LIN {X 0,Y 420.408,Z 179.012,A -85,B 0,C 180,E1 -10010.808,E2 -10010.808} C_VEL
LIN {X 0,Y 420.567,Z 173.267,A -85,B 0,C 180,E1 -10012.086,E2 -10012.086} C_VEL
LIN {X 0,Y 418.323,Z 161.696,A -85,B 0,C 180,E1 -10014.875,E2 -10014.875} C_VEL
LIN {X 0,Y 418.291,Z 161.388,A -85,B 0,C 180,E1 -10015.076,E2 -10015.076} C_VEL
LIN {X 0,Y 418.293,Z 161.379,A -85,B 0,C 180,E1 -10018.063,E2 -10018.063} C_VEL
LIN {X 0,Y 418.212,Z 161.381,A -85,B 0,C 180,E1 -10021.396,E2 -10021.396} C_VEL
LIN {X 0,Y 418.266,Z 161.374,A -85,B 0,C 180,E1 -10024.58,E2 -10024.58} C_VEL
LIN {X 0,Y 418.226,Z 161.39,A -85,B 0,C 180,E1 -10027.833,E2 -10027.833} C_VEL
LIN {X 0,Y 418.221,Z 161.38,A -85,B 0,C 180,E1 -10030.948,E2 -10030.948} C_VEL
LIN {X 0,Y 418.208,Z 161.391,A -85,B 0,C 180,E1 -10033.729,E2 -10033.729} C_VEL
LIN {X 0,Y 418.206,Z 161.372,A -85,B 0,C 180,E1 -10036.448,E2 -10036.448} C_VEL
LIN {X 0,Y 418.222,Z 161.384,A -85,B 0,C 180,E1 -10039.129,E2 -10039.129} C_VEL
LIN {X 0,Y 418.227,Z 161.383,A -85,B 0,C 180,E1 -10042.166,E2 -10042.166} C_VEL
LIN {X 0,Y 418.262,Z 161.354,A -85,B 0,C 180,E1 -10045.419,E2 -10045.419} C_VEL
LIN {X 0,Y 418.208,Z 161.389,A -85,B 0,C 180,E1 -10048.603,E2 -10048.603} C_VEL
LIN {X 0,Y 418.287,Z 161.376,A -85,B 0,C 180,E1 -10051.936,E2 -10051.936} C_VEL
LIN {X 0,Y 418.285,Z 161.379,A -85,B 0,C 180,E1 -10055.162,E2 -10055.162} C_VEL
LIN {X 0,Y 418.228,Z 161.382,A -85,B 0,C 180,E1 -10058.303,E2 -10058.303} C_VEL
LIN {X 0,Y 418.278,Z 161.382,A -85,B 0,C 180,E1 -10061.383,E2 -10061.383} C_VEL
LIN {X 0,Y 418.296,Z 161.369,A -85,B 0,C 180,E1 -10064.406,E2 -10064.406} C_VEL
LIN {X 0,Y 418.349,Z 161.372,A -85,B 0,C 180,E1 -10067.385,E2 -10067.385} C_VEL
LIN {X 0,Y 418.334,Z 161.361,A -85,B 0,C 180,E1 -10070.328,E2 -10070.328} C_VEL
LIN {X 0,Y 418.507,Z 161.348,A -85,B 0,C 180,E1 -10072.279,E2 -10072.279} C_VEL
LIN {X 0,Y 418.502,Z 161.352,A -85,B 0,C 180,E1 -10074.217,E2 -10074.217} C_VEL
LIN {X 0,Y 418.534,Z 161.342,A -85,B 0,C 180,E1 -10078.075,E2 -10078.075} C_VEL
LIN {X 0,Y 418.663,Z 161.333,A -85,B 0,C 180,E1 -10080,E2 -10080} C_VEL
LIN {X 0,Y 418.492,Z 161.352,A -85,B 0,C 180,E1 -10082.888,E2 -10082.888} C_VEL
LIN {X 0,Y 418.497,Z 161.352,A -85,B 0,C 180,E1 -10085.783,E2 -10085.783} C_VEL
LIN {X 0,Y 418.371,Z 161.368,A -85,B 0,C 180,E1 -10088.696,E2 -10088.696} C_VEL
LIN {X 0,Y 418.308,Z 161.37,A -85,B 0,C 180,E1 -10091.631,E2 -10091.631} C_VEL
LIN {X 0,Y 418.296,Z 161.377,A -85,B 0,C 180,E1 -10094.597,E2 -10094.597} C_VEL
LIN {X 0,Y 418.273,Z 161.374,A -85,B 0,C 180,E1 -10097.604,E2 -10097.604} C_VEL
LIN {X 0,Y 418.244,Z 161.384,A -85,B 0,C 180,E1 -10100.663,E2 -10100.663} C_VEL
LIN {X 0,Y 418.269,Z 161.374,A -85,B 0,C 180,E1 -10103.782,E2 -10103.782} C_VEL
LIN {X 0,Y 418.306,Z 161.382,A -85,B 0,C 180,E1 -10107.071,E2 -10107.071} C_VEL
LIN {X 0,Y 418.24,Z 161.38,A -85,B 0,C 180,E1 -10110.273,E2 -10110.273} C_VEL
LIN {X 0,Y 418.243,Z 161.38,A -85,B 0,C 180,E1 -10113.678,E2 -10113.678} C_VEL
LIN {X 0,Y 418.236,Z 161.366,A -85,B 0,C 180,E1 -10117.225,E2 -10117.225} C_VEL
LIN {X 0,Y 418.24,Z 161.384,A -85,B 0,C 180,E1 -10119.683,E2 -10119.683} C_VEL
LIN {X 0,Y 418.22,Z 161.386,A -85,B 0,C 180,E1 -10122.321,E2 -10122.321} C_VEL
LIN {X 0,Y 418.233,Z 161.39,A -85,B 0,C 180,E1 -10125.109,E2 -10125.109} C_VEL
LIN {X 0,Y 418.221,Z 161.386,A -85,B 0,C 180,E1 -10127.765,E2 -10127.765} C_VEL
LIN {X 0,Y 418.236,Z 161.372,A -85,B 0,C 180,E1 -10131.557,E2 -10131.557} C_VEL
LIN {X 0,Y 418.258,Z 161.379,A -85,B 0,C 180,E1 -10135.159,E2 -10135.159} C_VEL
LIN {X 0,Y 418.245,Z 161.387,A -85,B 0,C 180,E1 -10137.472,E2 -10137.472} C_VEL
LIN {X 0,Y 418.263,Z 161.386,A -85,B 0,C 180,E1 -10140.897,E2 -10140.897} C_VEL
LIN {X 0,Y 418.285,Z 161.441,A -85,B 0,C 180,E1 -10143.695,E2 -10143.695} C_VEL
LIN {X 0,Y 420.231,Z 171.346,A -85,B 0,C 180,E1 -10146.074,E2 -10146.074} C_VEL
LIN {X 0,Y 420.944,Z 175.757,A -85,B 0,C 180,E1 -10147.079,E2 -10147.079} C_VEL
LIN {X 0,Y 420.015,Z 190.491,A -85,B 0,C 180,E1 -10150.21,E2 -10150.21} C_VEL
LIN {X 0,Y 419.851,Z 194.089,A -85,B 0,C 180,E1 -10150.917,E2 -10150.917} C_VEL
LIN {X 0,Y 422.242,Z 207.63,A -85,B 0,C 180,E1 -10151.3,E2 -10151.3} C_VEL
LIN {X 0,Y 423.878,Z 217.834,A -85,B 0,C 180,E1 -10151.553,E2 -10151.553} C_VEL
LIN {X 0,Y 422.982,Z 301.78,A -85,B 0,C 180,E1 -10153.003,E2 -10153.003} C_VEL
LIN {X 0,Y 422.43,Z 315.009,A -85,B 0,C 180,E1 -10153.415,E2 -10153.415} C_VEL
LIN {X 0,Y 421.891,Z 327.144,A -85,B 0,C 180,E1 -10153.984,E2 -10153.984} C_VEL
LIN {X 0,Y 421.162,Z 339.385,A -85,B 0,C 180,E1 -10154.762,E2 -10154.762} C_VEL
LIN {X 0,Y 420.427,Z 350.645,A -85,B 0,C 180,E1 -10155.696,E2 -10155.696} C_VEL
LIN {X 0,Y 419.714,Z 361.373,A -85,B 0,C 180,E1 -10156.812,E2 -10156.812} C_VEL
LIN {X 0,Y 419.06,Z 369.887,A -85,B 0,C 180,E1 -10157.899,E2 -10157.899} C_VEL
LIN {X 0,Y 418.446,Z 377.741,A -85,B 0,C 180,E1 -10159.108,E2 -10159.108} C_VEL
LIN {X 0,Y 417.882,Z 385.409,A -85,B 0,C 180,E1 -10160.562,E2 -10160.562} C_VEL
LIN {X 0,Y 417.432,Z 392.477,A -85,B 0,C 180,E1 -10162.259,E2 -10162.259} C_VEL
LIN {X 0,Y 417.239,Z 396.897,A -85,B 0,C 180,E1 -10163.618,E2 -10163.618} C_VEL
LIN {X 0,Y 417.146,Z 400.769,A -85,B 0,C 180,E1 -10165.167,E2 -10165.167} C_VEL
LIN {X 0,Y 417.016,Z 402.62,A -85,B 0,C 180,E1 -10166.134,E2 -10166.134} C_VEL
LIN {X 0,Y 417.031,Z 404.999,A -85,B 0,C 180,E1 -10168.068,E2 -10168.068} C_VEL
LIN {X 0,Y 416.982,Z 405.818,A -85,B 0,C 180,E1 -10170,E2 -10170} C_VEL
LIN {X 0,Y 417.031,Z 404.997,A -85,B 0,C 180,E1 -10171.931,E2 -10171.931} C_VEL
LIN {X 0,Y 417.016,Z 402.616,A -85,B 0,C 180,E1 -10173.865,E2 -10173.865} C_VEL
LIN {X 0,Y 417.167,Z 399.693,A -85,B 0,C 180,E1 -10175.316,E2 -10175.316} C_VEL
LIN {X 0,Y 417.316,Z 395.735,A -85,B 0,C 180,E1 -10176.77,E2 -10176.77} C_VEL
LIN {X 0,Y 417.616,Z 389.647,A -85,B 0,C 180,E1 -10178.467,E2 -10178.467} C_VEL
LIN {X 0,Y 418.044,Z 382.993,A -85,B 0,C 180,E1 -10179.922,E2 -10179.922} C_VEL
LIN {X 0,Y 418.643,Z 374.734,A -85,B 0,C 180,E1 -10181.376,E2 -10181.376} C_VEL
LIN {X 0,Y 419.337,Z 366.267,A -85,B 0,C 180,E1 -10182.584,E2 -10182.584} C_VEL
LIN {X 0,Y 420.064,Z 355.745,A -85,B 0,C 180,E1 -10183.798,E2 -10183.798} C_VEL
LIN {X 0,Y 420.83,Z 344.015,A -85,B 0,C 180,E1 -10184.878,E2 -10184.878} C_VEL
LIN {X 0,Y 421.563,Z 332.157,A -85,B 0,C 180,E1 -10185.718,E2 -10185.718} C_VEL
LIN {X 0,Y 422.237,Z 319.815,A -85,B 0,C 180,E1 -10186.374,E2 -10186.374} C_VEL
LIN {X 0,Y 422.762,Z 307.137,A -85,B 0,C 180,E1 -10186.85,E2 -10186.85} C_VEL
LIN {X 0,Y 423.082,Z 293.853,A -85,B 0,C 180,E1 -10187.148,E2 -10187.148} C_VEL
LIN {X 0,Y 423.755,Z 216.699,A -85,B 0,C 180,E1 -10188.465,E2 -10188.465} C_VEL
LIN {X 0,Y 419.861,Z 194.269,A -85,B 0,C 180,E1 -10189.059,E2 -10189.059} C_VEL
LIN {X 0,Y 419.935,Z 191.573,A -85,B 0,C 180,E1 -10189.554,E2 -10189.554} C_VEL
LIN {X 0,Y 420.92,Z 177.278,A -85,B 0,C 180,E1 -10192.582,E2 -10192.582} C_VEL
LIN {X 0,Y 420.491,Z 172.503,A -85,B 0,C 180,E1 -10193.648,E2 -10193.648} C_VEL
LIN {X 0,Y 418.304,Z 161.56,A -85,B 0,C 180,E1 -10196.236,E2 -10196.236} C_VEL
LIN {X 0,Y 418.257,Z 161.387,A -85,B 0,C 180,E1 -10199.161,E2 -10199.161} C_VEL
LIN {X 0,Y 418.254,Z 161.384,A -85,B 0,C 180,E1 -10202.843,E2 -10202.843} C_VEL
LIN {X 0,Y 418.239,Z 161.386,A -85,B 0,C 180,E1 -10206.237,E2 -10206.237} C_VEL
LIN {X 0,Y 418.223,Z 161.386,A -85,B 0,C 180,E1 -10209.683,E2 -10209.683} C_VEL
LIN {X 0,Y 418.217,Z 161.386,A -85,B 0,C 180,E1 -10212.319,E2 -10212.319} C_VEL
LIN {X 0,Y 418.23,Z 161.39,A -85,B 0,C 180,E1 -10215.108,E2 -10215.108} C_VEL
LIN {X 0,Y 418.233,Z 161.384,A -85,B 0,C 180,E1 -10217.766,E2 -10217.766} C_VEL
LIN {X 0,Y 418.238,Z 161.386,A -85,B 0,C 180,E1 -10220.62,E2 -10220.62} C_VEL
LIN {X 0,Y 418.234,Z 161.365,A -85,B 0,C 180,E1 -10223.975,E2 -10223.975} C_VEL
LIN {X 0,Y 418.248,Z 161.388,A -85,B 0,C 180,E1 -10227.155,E2 -10227.155} C_VEL
LIN {X 0,Y 418.259,Z 161.38,A -85,B 0,C 180,E1 -10230.895,E2 -10230.895} C_VEL
LIN {X 0,Y 418.258,Z 161.382,A -85,B 0,C 180,E1 -10234.095,E2 -10234.095} C_VEL
LIN {X 0,Y 418.22,Z 161.387,A -85,B 0,C 180,E1 -10237.263,E2 -10237.263} C_VEL
LIN {X 0,Y 418.271,Z 161.382,A -85,B 0,C 180,E1 -10240.364,E2 -10240.364} C_VEL
LIN {X 0,Y 418.304,Z 161.374,A -85,B 0,C 180,E1 -10243.404,E2 -10243.404} C_VEL
LIN {X 0,Y 418.344,Z 161.368,A -85,B 0,C 180,E1 -10246.994,E2 -10246.994} C_VEL
LIN {X 0,Y 418.332,Z 161.37,A -85,B 0,C 180,E1 -10250.328,E2 -10250.328} C_VEL
LIN {X 0,Y 418.477,Z 161.352,A -85,B 0,C 180,E1 -10253.249,E2 -10253.249} C_VEL
LIN {X 0,Y 418.324,Z 161.364,A -85,B 0,C 180,E1 -10255.181,E2 -10255.181} C_VEL
LIN {X 0,Y 418.53,Z 161.348,A -85,B 0,C 180,E1 -10258.075,E2 -10258.075} C_VEL
LIN {X 0,Y 418.659,Z 161.333,A -85,B 0,C 180,E1 -10260,E2 -10260} C_VEL
LIN {X 0,Y 418.487,Z 161.349,A -85,B 0,C 180,E1 -10262.888,E2 -10262.888} C_VEL
LIN {X 0,Y 418.478,Z 161.354,A -85,B 0,C 180,E1 -10266.751,E2 -10266.751} C_VEL
LIN {X 0,Y 418.388,Z 161.357,A -85,B 0,C 180,E1 -10268.695,E2 -10268.695} C_VEL
LIN {X 0,Y 418.304,Z 161.374,A -85,B 0,C 180,E1 -10271.631,E2 -10271.631} C_VEL
LIN {X 0,Y 418.291,Z 161.373,A -85,B 0,C 180,E1 -10274.598,E2 -10274.598} C_VEL
LIN {X 0,Y 418.277,Z 161.377,A -85,B 0,C 180,E1 -10277.604,E2 -10277.604} C_VEL
LIN {X 0,Y 418.239,Z 161.381,A -85,B 0,C 180,E1 -10280.664,E2 -10280.664} C_VEL
LIN {X 0,Y 418.278,Z 161.378,A -85,B 0,C 180,E1 -10283.782,E2 -10283.782} C_VEL
LIN {X 0,Y 418.301,Z 161.371,A -85,B 0,C 180,E1 -10287.071,E2 -10287.071} C_VEL
LIN {X 0,Y 418.235,Z 161.39,A -85,B 0,C 180,E1 -10290.273,E2 -10290.273} C_VEL
LIN {X 0,Y 418.24,Z 161.372,A -85,B 0,C 180,E1 -10293.678,E2 -10293.678} C_VEL
LIN {X 0,Y 418.232,Z 161.376,A -85,B 0,C 180,E1 -10297.225,E2 -10297.225} C_VEL
LIN {X 0,Y 418.241,Z 161.387,A -85,B 0,C 180,E1 -10299.683,E2 -10299.683} C_VEL
LIN {X 0,Y 418.222,Z 161.374,A -85,B 0,C 180,E1 -10302.322,E2 -10302.322} C_VEL
LIN {X 0,Y 418.229,Z 161.379,A -85,B 0,C 180,E1 -10305.11,E2 -10305.11} C_VEL
LIN {X 0,Y 418.234,Z 161.388,A -85,B 0,C 180,E1 -10307.768,E2 -10307.768} C_VEL
LIN {X 0,Y 418.24,Z 161.374,A -85,B 0,C 180,E1 -10310.622,E2 -10310.622} C_VEL
LIN {X 0,Y 418.24,Z 161.383,A -85,B 0,C 180,E1 -10313.977,E2 -10313.977} C_VEL
LIN {X 0,Y 418.255,Z 161.385,A -85,B 0,C 180,E1 -10317.157,E2 -10317.157} C_VEL
LIN {X 0,Y 418.267,Z 161.383,A -85,B 0,C 180,E1 -10320.897,E2 -10320.897} C_VEL
LIN {X 0,Y 418.269,Z 161.383,A -85,B 0,C 180,E1 -10324.097,E2 -10324.097} C_VEL
LIN {X 0,Y 418.289,Z 161.528,A -85,B 0,C 180,E1 -10325.164,E2 -10325.164} C_VEL
LIN {X 0,Y 420.482,Z 172.831,A -85,B 0,C 180,E1 -10327.911,E2 -10327.911} C_VEL
LIN {X 0,Y 420.548,Z 176.275,A -85,B 0,C 180,E1 -10328.687,E2 -10328.687} C_VEL
LIN {X 0,Y 419.948,Z 186.936,A -85,B 0,C 180,E1 -10330.972,E2 -10330.972} C_VEL
LIN {X 0,Y 421.24,Z 194.005,A -85,B 0,C 180,E1 -10331.195,E2 -10331.195} C_VEL
LIN {X 0,Y 423.914,Z 208.785,A -85,B 0,C 180,E1 -10331.578,E2 -10331.578} C_VEL
LIN {X 0,Y 423.001,Z 294.776,A -85,B 0,C 180,E1 -10333.067,E2 -10333.067} C_VEL
LIN {X 0,Y 422.592,Z 307.097,A -85,B 0,C 180,E1 -10333.454,E2 -10333.454} C_VEL
LIN {X 0,Y 421.954,Z 319.914,A -85,B 0,C 180,E1 -10334.049,E2 -10334.049} C_VEL
LIN {X 0,Y 421.314,Z 331.29,A -85,B 0,C 180,E1 -10334.769,E2 -10334.769} C_VEL
LIN {X 0,Y 420.637,Z 342.748,A -85,B 0,C 180,E1 -10335.712,E2 -10335.712} C_VEL
LIN {X 0,Y 419.925,Z 353.455,A -85,B 0,C 180,E1 -10336.819,E2 -10336.819} C_VEL
LIN {X 0,Y 419.231,Z 362.024,A -85,B 0,C 180,E1 -10337.905,E2 -10337.905} C_VEL
LIN {X 0,Y 418.653,Z 369.918,A -85,B 0,C 180,E1 -10339.115,E2 -10339.115} C_VEL
LIN {X 0,Y 418.129,Z 376.948,A -85,B 0,C 180,E1 -10340.425,E2 -10340.425} C_VEL
LIN {X 0,Y 417.298,Z 380.14,A -85,B 0,C 180,E1 -10341.099,E2 -10341.099} C_VEL
LIN {X 0,Y 414.13,Z 384.851,A -85,B 0,C 180,E1 -10342.219,E2 -10342.219} C_VEL
LIN {X 0,Y 410.989,Z 388.898,A -85,B 0,C 180,E1 -10343.402,E2 -10343.402} C_VEL
LIN {X 0,Y 410.217,Z 390.994,A -85,B 0,C 180,E1 -10344.167,E2 -10344.167} C_VEL
LIN {X 0,Y 410.126,Z 393.124,A -85,B 0,C 180,E1 -10345.085,E2 -10345.085} C_VEL
LIN {X 0,Y 409.982,Z 394.993,A -85,B 0,C 180,E1 -10346.069,E2 -10346.069} C_VEL
LIN {X 0,Y 409.952,Z 396.401,A -85,B 0,C 180,E1 -10347.052,E2 -10347.052} C_VEL
LIN {X 0,Y 409.971,Z 397.401,A -85,B 0,C 180,E1 -10348.036,E2 -10348.036} C_VEL
LIN {X 0,Y 409.907,Z 398.253,A -85,B 0,C 180,E1 -10350,E2 -10350} C_VEL
LIN {X 0,Y 409.92,Z 398.064,A -85,B 0,C 180,E1 -10350.983,E2 -10350.983} C_VEL
LIN {X 0,Y 409.971,Z 397.477,A -85,B 0,C 180,E1 -10351.965,E2 -10351.965} C_VEL
LIN {X 0,Y 409.979,Z 395.145,A -85,B 0,C 180,E1 -10353.932,E2 -10353.932} C_VEL
LIN {X 0,Y 410.166,Z 392.267,A -85,B 0,C 180,E1 -10355.408,E2 -10355.408} C_VEL
LIN {X 0,Y 410.347,Z 388.366,A -85,B 0,C 180,E1 -10356.886,E2 -10356.886} C_VEL
LIN {X 0,Y 410.618,Z 383.335,A -85,B 0,C 180,E1 -10358.365,E2 -10358.365} C_VEL
LIN {X 0,Y 411.124,Z 377.002,A -85,B 0,C 180,E1 -10359.843,E2 -10359.843} C_VEL
LIN {X 0,Y 411.71,Z 369.077,A -85,B 0,C 180,E1 -10361.321,E2 -10361.321} C_VEL
LIN {X 0,Y 412.541,Z 359.221,A -85,B 0,C 180,E1 -10362.795,E2 -10362.795} C_VEL
LIN {X 0,Y 413.278,Z 349.771,A -85,B 0,C 180,E1 -10363.929,E2 -10363.929} C_VEL
LIN {X 0,Y 413.976,Z 338.643,A -85,B 0,C 180,E1 -10365.005,E2 -10365.005} C_VEL
LIN {X 0,Y 414.802,Z 327.443,A -85,B 0,C 180,E1 -10365.855,E2 -10365.855} C_VEL
LIN {X 0,Y 415.4,Z 316.084,A -85,B 0,C 180,E1 -10366.526,E2 -10366.526} C_VEL
LIN {X 0,Y 415.978,Z 303.133,A -85,B 0,C 180,E1 -10367.071,E2 -10367.071} C_VEL
LIN {X 0,Y 416.339,Z 289.288,A -85,B 0,C 180,E1 -10367.435,E2 -10367.435} C_VEL
LIN {X 0,Y 417.045,Z 208.536,A -85,B 0,C 180,E1 -10368.841,E2 -10368.841} C_VEL
LIN {X 0,Y 413.049,Z 187.174,A -85,B 0,C 180,E1 -10369.443,E2 -10369.443} C_VEL
LIN {X 0,Y 413.47,Z 180.22,A -85,B 0,C 180,E1 -10370.913,E2 -10370.913} C_VEL
LIN {X 0,Y 413.742,Z 175.616,A -85,B 0,C 180,E1 -10371.944,E2 -10371.944} C_VEL
LIN {X 0,Y 411.652,Z 164.315,A -85,B 0,C 180,E1 -10374.687,E2 -10374.687} C_VEL
LIN {X 0,Y 411.241,Z 162.288,A -85,B 0,C 180,E1 -10375.273,E2 -10375.273} C_VEL
LIN {X 0,Y 411.26,Z 162.258,A -85,B 0,C 180,E1 -10377.477,E2 -10377.477} C_VEL
LIN {X 0,Y 411.19,Z 162.257,A -85,B 0,C 180,E1 -10380.847,E2 -10380.847} C_VEL
LIN {X 0,Y 411.206,Z 162.255,A -85,B 0,C 180,E1 -10384.333,E2 -10384.333} C_VEL
LIN {X 0,Y 411.191,Z 162.266,A -85,B 0,C 180,E1 -10387.973,E2 -10387.973} C_VEL
LIN {X 0,Y 411.162,Z 162.258,A -85,B 0,C 180,E1 -10391.228,E2 -10391.228} C_VEL
LIN {X 0,Y 411.174,Z 162.262,A -85,B 0,C 180,E1 -10394.49,E2 -10394.49} C_VEL
LIN {X 0,Y 411.175,Z 162.256,A -85,B 0,C 180,E1 -10398.194,E2 -10398.194} C_VEL
LIN {X 0,Y 411.219,Z 162.259,A -85,B 0,C 180,E1 -10400.776,E2 -10400.776} C_VEL
LIN {X 0,Y 411.195,Z 162.233,A -85,B 0,C 180,E1 -10404.471,E2 -10404.471} C_VEL
LIN {X 0,Y 411.204,Z 162.251,A -85,B 0,C 180,E1 -10406.873,E2 -10406.873} C_VEL
LIN {X 0,Y 411.229,Z 162.256,A -85,B 0,C 180,E1 -10410.644,E2 -10410.644} C_VEL
LIN {X 0,Y 411.232,Z 162.255,A -85,B 0,C 180,E1 -10413.619,E2 -10413.619} C_VEL
LIN {X 0,Y 411.19,Z 162.259,A -85,B 0,C 180,E1 -10416.852,E2 -10416.852} C_VEL
LIN {X 0,Y 411.21,Z 162.264,A -85,B 0,C 180,E1 -10420.05,E2 -10420.05} C_VEL
LIN {X 0,Y 411.258,Z 162.252,A -85,B 0,C 180,E1 -10423.131,E2 -10423.131} C_VEL
LIN {X 0,Y 411.3,Z 162.247,A -85,B 0,C 180,E1 -10426.896,E2 -10426.896} C_VEL
LIN {X 0,Y 411.286,Z 162.24,A -85,B 0,C 180,E1 -10430.161,E2 -10430.161} C_VEL
LIN {X 0,Y 411.476,Z 162.225,A -85,B 0,C 180,E1 -10432.146,E2 -10432.146} C_VEL
LIN {X 0,Y 411.464,Z 162.229,A -85,B 0,C 180,E1 -10434.118,E2 -10434.118} C_VEL
LIN {X 0,Y 411.503,Z 162.217,A -85,B 0,C 180,E1 -10438.042,E2 -10438.042} C_VEL
LIN {X 0,Y 411.632,Z 162.209,A -85,B 0,C 180,E1 -10440,E2 -10440} C_VEL
LIN {X 0,Y 411.449,Z 162.23,A -85,B 0,C 180,E1 -10442.937,E2 -10442.937} C_VEL
LIN {X 0,Y 411.458,Z 162.228,A -85,B 0,C 180,E1 -10445.882,E2 -10445.882} C_VEL
LIN {X 0,Y 411.312,Z 162.248,A -85,B 0,C 180,E1 -10448.846,E2 -10448.846} C_VEL
LIN {X 0,Y 411.277,Z 162.247,A -85,B 0,C 180,E1 -10451.833,E2 -10451.833} C_VEL
LIN {X 0,Y 411.253,Z 162.256,A -85,B 0,C 180,E1 -10454.853,E2 -10454.853} C_VEL
LIN {X 0,Y 411.239,Z 162.249,A -85,B 0,C 180,E1 -10457.916,E2 -10457.916} C_VEL
LIN {X 0,Y 411.19,Z 162.266,A -85,B 0,C 180,E1 -10461.034,E2 -10461.034} C_VEL
LIN {X 0,Y 411.206,Z 162.253,A -85,B 0,C 180,E1 -10464.217,E2 -10464.217} C_VEL
LIN {X 0,Y 411.254,Z 162.256,A -85,B 0,C 180,E1 -10467.478,E2 -10467.478} C_VEL
LIN {X 0,Y 411.185,Z 162.263,A -85,B 0,C 180,E1 -10470.848,E2 -10470.848} C_VEL
LIN {X 0,Y 411.2,Z 162.256,A -85,B 0,C 180,E1 -10474.334,E2 -10474.334} C_VEL
LIN {X 0,Y 411.188,Z 162.251,A -85,B 0,C 180,E1 -10477.975,E2 -10477.975} C_VEL
LIN {X 0,Y 411.157,Z 162.269,A -85,B 0,C 180,E1 -10481.228,E2 -10481.228} C_VEL
LIN {X 0,Y 411.173,Z 162.265,A -85,B 0,C 180,E1 -10484.491,E2 -10484.491} C_VEL
LIN {X 0,Y 411.162,Z 162.266,A -85,B 0,C 180,E1 -10488.193,E2 -10488.193} C_VEL
LIN {X 0,Y 411.181,Z 162.255,A -85,B 0,C 180,E1 -10490.772,E2 -10490.772} C_VEL
LIN {X 0,Y 411.196,Z 162.267,A -85,B 0,C 180,E1 -10494.472,E2 -10494.472} C_VEL
LIN {X 0,Y 411.207,Z 162.258,A -85,B 0,C 180,E1 -10496.874,E2 -10496.874} C_VEL
LIN {X 0,Y 411.212,Z 162.265,A -85,B 0,C 180,E1 -10500.65,E2 -10500.65} C_VEL
LIN {X 0,Y 411.273,Z 162.44,A -85,B 0,C 180,E1 -10503.489,E2 -10503.489} C_VEL
LIN {X 0,Y 413.754,Z 175.101,A -85,B 0,C 180,E1 -10506.527,E2 -10506.527} C_VEL
LIN {X 0,Y 413.998,Z 178.443,A -85,B 0,C 180,E1 -10507.282,E2 -10507.282} C_VEL
LIN {X 0,Y 412.963,Z 194.027,A -85,B 0,C 180,E1 -10510.587,E2 -10510.587} C_VEL
LIN {X 0,Y 416.04,Z 211.615,A -85,B 0,C 180,E1 -10511.083,E2 -10511.083} C_VEL
LIN {X 0,Y 417.134,Z 219.006,A -85,B 0,C 180,E1 -10511.266,E2 -10511.266} C_VEL
LIN {X 0,Y 416.213,Z 301.727,A -85,B 0,C 180,E1 -10512.718,E2 -10512.718} C_VEL
LIN {X 0,Y 415.636,Z 314.952,A -85,B 0,C 180,E1 -10513.136,E2 -10513.136} C_VEL
LIN {X 0,Y 415.081,Z 327.085,A -85,B 0,C 180,E1 -10513.714,E2 -10513.714} C_VEL
LIN {X 0,Y 414.307,Z 339.324,A -85,B 0,C 180,E1 -10514.504,E2 -10514.504} C_VEL
LIN {X 0,Y 413.541,Z 350.579,A -85,B 0,C 180,E1 -10515.452,E2 -10515.452} C_VEL
LIN {X 0,Y 412.778,Z 361.311,A -85,B 0,C 180,E1 -10516.586,E2 -10516.586} C_VEL
LIN {X 0,Y 412.102,Z 369.825,A -85,B 0,C 180,E1 -10517.691,E2 -10517.691} C_VEL
LIN {X 0,Y 411.428,Z 377.677,A -85,B 0,C 180,E1 -10518.92,E2 -10518.92} C_VEL
LIN {X 0,Y 410.859,Z 385.345,A -85,B 0,C 180,E1 -10520.399,E2 -10520.399} C_VEL
LIN {X 0,Y 410.378,Z 392.413,A -85,B 0,C 180,E1 -10522.125,E2 -10522.125} C_VEL
LIN {X 0,Y 410.133,Z 397.276,A -85,B 0,C 180,E1 -10523.661,E2 -10523.661} C_VEL
LIN {X 0,Y 410.058,Z 400.705,A -85,B 0,C 180,E1 -10525.084,E2 -10525.084} C_VEL
LIN {X 0,Y 409.936,Z 402.556,A -85,B 0,C 180,E1 -10526.067,E2 -10526.067} C_VEL
LIN {X 0,Y 409.927,Z 404.935,A -85,B 0,C 180,E1 -10528.035,E2 -10528.035} C_VEL
LIN {X 0,Y 409.918,Z 405.539,A -85,B 0,C 180,E1 -10529.017,E2 -10529.017} C_VEL
LIN {X 0,Y 409.906,Z 405.753,A -85,B 0,C 180,E1 -10530,E2 -10530} C_VEL
LIN {X 0,Y 409.918,Z 405.537,A -85,B 0,C 180,E1 -10530.982,E2 -10530.982} C_VEL
LIN {X 0,Y 409.927,Z 404.932,A -85,B 0,C 180,E1 -10531.965,E2 -10531.965} C_VEL
LIN {X 0,Y 409.936,Z 402.55,A -85,B 0,C 180,E1 -10533.932,E2 -10533.932} C_VEL
LIN {X 0,Y 410.086,Z 399.627,A -85,B 0,C 180,E1 -10535.408,E2 -10535.408} C_VEL
LIN {X 0,Y 410.251,Z 395.669,A -85,B 0,C 180,E1 -10536.887,E2 -10536.887} C_VEL
LIN {X 0,Y 410.562,Z 389.58,A -85,B 0,C 180,E1 -10538.614,E2 -10538.614} C_VEL
LIN {X 0,Y 411.017,Z 382.926,A -85,B 0,C 180,E1 -10540.093,E2 -10540.093} C_VEL
LIN {X 0,Y 411.644,Z 374.667,A -85,B 0,C 180,E1 -10541.572,E2 -10541.572} C_VEL
LIN {X 0,Y 412.404,Z 366.2,A -85,B 0,C 180,E1 -10542.799,E2 -10542.799} C_VEL
LIN {X 0,Y 413.104,Z 356.439,A -85,B 0,C 180,E1 -10543.954,E2 -10543.954} C_VEL
LIN {X 0,Y 413.852,Z 345.373,A -85,B 0,C 180,E1 -10545.008,E2 -10545.008} C_VEL
LIN {X 0,Y 414.602,Z 334.012,A -85,B 0,C 180,E1 -10545.862,E2 -10545.862} C_VEL
LIN {X 0,Y 415.304,Z 322.345,A -85,B 0,C 180,E1 -10546.529,E2 -10546.529} C_VEL
LIN {X 0,Y 415.899,Z 308.893,A -85,B 0,C 180,E1 -10547.073,E2 -10547.073} C_VEL
LIN {X 0,Y 416.284,Z 295.555,A -85,B 0,C 180,E1 -10547.405,E2 -10547.405} C_VEL
LIN {X 0,Y 417.099,Z 218,A -85,B 0,C 180,E1 -10548.745,E2 -10548.745} C_VEL
LIN {X 0,Y 412.956,Z 194.35,A -85,B 0,C 180,E1 -10549.381,E2 -10549.381} C_VEL
LIN {X 0,Y 412.957,Z 192.697,A -85,B 0,C 180,E1 -10549.639,E2 -10549.639} C_VEL
LIN {X 0,Y 413.98,Z 178.402,A -85,B 0,C 180,E1 -10552.718,E2 -10552.718} C_VEL
LIN {X 0,Y 413.603,Z 174.093,A -85,B 0,C 180,E1 -10553.696,E2 -10553.696} C_VEL
LIN {X 0,Y 411.27,Z 162.413,A -85,B 0,C 180,E1 -10556.511,E2 -10556.511} C_VEL
LIN {X 0,Y 411.195,Z 162.263,A -85,B 0,C 180,E1 -10559.712,E2 -10559.712} C_VEL
LIN {X 0,Y 411.203,Z 162.258,A -85,B 0,C 180,E1 -10563.155,E2 -10563.155} C_VEL
LIN {X 0,Y 411.187,Z 162.266,A -85,B 0,C 180,E1 -10566.551,E2 -10566.551} C_VEL
LIN {X 0,Y 411.19,Z 162.262,A -85,B 0,C 180,E1 -10569.724,E2 -10569.724} C_VEL
LIN {X 0,Y 411.165,Z 162.266,A -85,B 0,C 180,E1 -10573.133,E2 -10573.133} C_VEL
LIN {X 0,Y 411.161,Z 162.264,A -85,B 0,C 180,E1 -10575.88,E2 -10575.88} C_VEL
LIN {X 0,Y 411.156,Z 162.269,A -85,B 0,C 180,E1 -10578.771,E2 -10578.771} C_VEL
LIN {X 0,Y 411.184,Z 162.25,A -85,B 0,C 180,E1 -10582.025,E2 -10582.025} C_VEL
LIN {X 0,Y 411.196,Z 162.257,A -85,B 0,C 180,E1 -10585.665,E2 -10585.665} C_VEL
LIN {X 0,Y 411.179,Z 162.263,A -85,B 0,C 180,E1 -10589.151,E2 -10589.151} C_VEL
LIN {X 0,Y 411.249,Z 162.256,A -85,B 0,C 180,E1 -10592.522,E2 -10592.522} C_VEL
LIN {X 0,Y 411.2,Z 162.252,A -85,B 0,C 180,E1 -10595.783,E2 -10595.783} C_VEL
LIN {X 0,Y 411.185,Z 162.267,A -85,B 0,C 180,E1 -10598.965,E2 -10598.965} C_VEL
LIN {X 0,Y 411.234,Z 162.249,A -85,B 0,C 180,E1 -10602.084,E2 -10602.084} C_VEL
LIN {X 0,Y 411.25,Z 162.257,A -85,B 0,C 180,E1 -10605.147,E2 -10605.147} C_VEL
LIN {X 0,Y 411.288,Z 162.245,A -85,B 0,C 180,E1 -10608.167,E2 -10608.167} C_VEL
LIN {X 0,Y 411.429,Z 162.235,A -85,B 0,C 180,E1 -10612.189,E2 -10612.189} C_VEL
LIN {X 0,Y 411.458,Z 162.228,A -85,B 0,C 180,E1 -10614.118,E2 -10614.118} C_VEL
LIN {X 0,Y 411.499,Z 162.224,A -85,B 0,C 180,E1 -10618.043,E2 -10618.043} C_VEL
LIN {X 0,Y 411.628,Z 162.209,A -85,B 0,C 180,E1 -10620,E2 -10620} C_VEL
LIN {X 0,Y 411.444,Z 162.226,A -85,B 0,C 180,E1 -10622.937,E2 -10622.937} C_VEL
LIN {X 0,Y 411.446,Z 162.229,A -85,B 0,C 180,E1 -10626.867,E2 -10626.867} C_VEL
LIN {X 0,Y 411.342,Z 162.233,A -85,B 0,C 180,E1 -10628.846,E2 -10628.846} C_VEL
LIN {X 0,Y 411.272,Z 162.251,A -85,B 0,C 180,E1 -10631.833,E2 -10631.833} C_VEL
LIN {X 0,Y 411.248,Z 162.248,A -85,B 0,C 180,E1 -10634.853,E2 -10634.853} C_VEL
LIN {X 0,Y 411.242,Z 162.255,A -85,B 0,C 180,E1 -10637.916,E2 -10637.916} C_VEL
LIN {X 0,Y 411.186,Z 162.257,A -85,B 0,C 180,E1 -10641.035,E2 -10641.035} C_VEL
LIN {X 0,Y 411.218,Z 162.263,A -85,B 0,C 180,E1 -10644.216,E2 -10644.216} C_VEL
LIN {X 0,Y 411.249,Z 162.25,A -85,B 0,C 180,E1 -10647.479,E2 -10647.479} C_VEL
LIN {X 0,Y 411.18,Z 162.264,A -85,B 0,C 180,E1 -10650.849,E2 -10650.849} C_VEL
LIN {X 0,Y 411.197,Z 162.238,A -85,B 0,C 180,E1 -10654.335,E2 -10654.335} C_VEL
LIN {X 0,Y 411.187,Z 162.26,A -85,B 0,C 180,E1 -10657.975,E2 -10657.975} C_VEL
LIN {X 0,Y 411.157,Z 162.265,A -85,B 0,C 180,E1 -10661.229,E2 -10661.229} C_VEL
LIN {X 0,Y 411.169,Z 162.256,A -85,B 0,C 180,E1 -10664.492,E2 -10664.492} C_VEL
LIN {X 0,Y 411.172,Z 162.262,A -85,B 0,C 180,E1 -10668.196,E2 -10668.196} C_VEL
LIN {X 0,Y 411.206,Z 162.251,A -85,B 0,C 180,E1 -10670.776,E2 -10670.776} C_VEL
LIN {X 0,Y 411.195,Z 162.255,A -85,B 0,C 180,E1 -10674.472,E2 -10674.472} C_VEL
LIN {X 0,Y 411.204,Z 162.262,A -85,B 0,C 180,E1 -10676.874,E2 -10676.874} C_VEL
LIN {X 0,Y 411.231,Z 162.26,A -85,B 0,C 180,E1 -10680.645,E2 -10680.645} C_VEL
LIN {X 0,Y 411.236,Z 162.258,A -85,B 0,C 180,E1 -10683.62,E2 -10683.62} C_VEL
LIN {X 0,Y 411.239,Z 162.46,A -85,B 0,C 180,E1 -10684.926,E2 -10684.926} C_VEL
LIN {X 0,Y 413.303,Z 172.889,A -85,B 0,C 180,E1 -10687.506,E2 -10687.506} C_VEL
LIN {X 0,Y 413.725,Z 176.333,A -85,B 0,C 180,E1 -10688.318,E2 -10688.318} C_VEL
LIN {X 0,Y 413.052,Z 187.056,A -85,B 0,C 180,E1 -10690.647,E2 -10690.647} C_VEL
LIN {X 0,Y 415.677,Z 200.949,A -85,B 0,C 180,E1 -10691.057,E2 -10691.057} C_VEL
LIN {X 0,Y 417.194,Z 210.215,A -85,B 0,C 180,E1 -10691.294,E2 -10691.294} C_VEL
LIN {X 0,Y 416.213,Z 294.858,A -85,B 0,C 180,E1 -10692.782,E2 -10692.782} C_VEL
LIN {X 0,Y 415.805,Z 307.173,A -85,B 0,C 180,E1 -10693.176,E2 -10693.176} C_VEL
LIN {X 0,Y 415.154,Z 319.987,A -85,B 0,C 180,E1 -10693.781,E2 -10693.781} C_VEL
LIN {X 0,Y 414.47,Z 331.361,A -85,B 0,C 180,E1 -10694.511,E2 -10694.511} C_VEL
LIN {X 0,Y 413.789,Z 341.958,A -85,B 0,C 180,E1 -10695.387,E2 -10695.387} C_VEL
LIN {X 0,Y 413.106,Z 352.456,A -85,B 0,C 180,E1 -10696.473,E2 -10696.473} C_VEL
LIN {X 0,Y 412.288,Z 362.092,A -85,B 0,C 180,E1 -10697.698,E2 -10697.698} C_VEL
LIN {X 0,Y 411.648,Z 369.986,A -85,B 0,C 180,E1 -10698.927,E2 -10698.927} C_VEL
LIN {X 0,Y 411.067,Z 377.704,A -85,B 0,C 180,E1 -10700.405,E2 -10700.405} C_VEL
LIN {X 0,Y 410.523,Z 384.789,A -85,B 0,C 180,E1 -10702.129,E2 -10702.129} C_VEL
LIN {X 0,Y 410.291,Z 389.1,A -85,B 0,C 180,E1 -10703.466,E2 -10703.466} C_VEL
LIN {X 0,Y 410.217,Z 390.994,A -85,B 0,C 180,E1 -10704.167,E2 -10704.167} C_VEL
LIN {X 0,Y 409.48,Z 392.861,A -85,B 0,C 180,E1 -10704.945,E2 -10704.945} C_VEL
LIN {X 0,Y 406.508,Z 395.32,A -85,B 0,C 180,E1 -10706.227,E2 -10706.227} C_VEL
LIN {X 0,Y 404.017,Z 396.758,A -85,B 0,C 180,E1 -10707.279,E2 -10707.279} C_VEL
LIN {X 0,Y 402.939,Z 397.545,A -85,B 0,C 180,E1 -10708.101,E2 -10708.101} C_VEL
LIN {X 0,Y 402.847,Z 397.701,A -85,B 0,C 180,E1 -10708.381,E2 -10708.381} C_VEL
LIN {X 0,Y 402.832,Z 398.318,A -85,B 0,C 180,E1 -10710,E2 -10710} C_VEL
LIN {X 0,Y 402.848,Z 398.129,A -85,B 0,C 180,E1 -10711,E2 -10711} C_VEL
LIN {X 0,Y 402.869,Z 397.542,A -85,B 0,C 180,E1 -10712,E2 -10712} C_VEL
LIN {X 0,Y 402.901,Z 395.209,A -85,B 0,C 180,E1 -10714.001,E2 -10714.001} C_VEL
LIN {X 0,Y 403.092,Z 392.331,A -85,B 0,C 180,E1 -10715.503,E2 -10715.503} C_VEL
LIN {X 0,Y 403.285,Z 388.43,A -85,B 0,C 180,E1 -10717.007,E2 -10717.007} C_VEL
LIN {X 0,Y 403.592,Z 383.398,A -85,B 0,C 180,E1 -10718.512,E2 -10718.512} C_VEL
LIN {X 0,Y 404.113,Z 377.065,A -85,B 0,C 180,E1 -10720.016,E2 -10720.016} C_VEL
LIN {X 0,Y 404.719,Z 369.14,A -85,B 0,C 180,E1 -10721.52,E2 -10721.52} C_VEL
LIN {X 0,Y 405.616,Z 359.282,A -85,B 0,C 180,E1 -10723.018,E2 -10723.018} C_VEL
LIN {X 0,Y 406.349,Z 350.147,A -85,B 0,C 180,E1 -10724.137,E2 -10724.137} C_VEL
LIN {X 0,Y 407.021,Z 340.127,A -85,B 0,C 180,E1 -10725.139,E2 -10725.139} C_VEL
LIN {X 0,Y 407.824,Z 329.265,A -85,B 0,C 180,E1 -10726.005,E2 -10726.005} C_VEL
LIN {X 0,Y 408.557,Z 317.271,A -85,B 0,C 180,E1 -10726.746,E2 -10726.746} C_VEL
LIN {X 0,Y 409.142,Z 304.984,A -85,B 0,C 180,E1 -10727.301,E2 -10727.301} C_VEL
LIN {X 0,Y 409.557,Z 292.34,A -85,B 0,C 180,E1 -10727.669,E2 -10727.669} C_VEL
LIN {X 0,Y 410.325,Z 209.43,A -85,B 0,C 180,E1 -10729.146,E2 -10729.146} C_VEL
LIN {X 0,Y 406.157,Z 187.245,A -85,B 0,C 180,E1 -10729.786,E2 -10729.786} C_VEL
LIN {X 0,Y 406.223,Z 184.89,A -85,B 0,C 180,E1 -10730.244,E2 -10730.244} C_VEL
LIN {X 0,Y 406.788,Z 176.822,A -85,B 0,C 180,E1 -10732.072,E2 -10732.072} C_VEL
LIN {X 0,Y 404.591,Z 165.109,A -85,B 0,C 180,E1 -10734.969,E2 -10734.969} C_VEL
LIN {X 0,Y 404.208,Z 163.161,A -85,B 0,C 180,E1 -10735.549,E2 -10735.549} C_VEL
LIN {X 0,Y 404.197,Z 163.135,A -85,B 0,C 180,E1 -10737.999,E2 -10737.999} C_VEL
LIN {X 0,Y 404.14,Z 163.134,A -85,B 0,C 180,E1 -10741.558,E2 -10741.558} C_VEL
LIN {X 0,Y 404.185,Z 163.126,A -85,B 0,C 180,E1 -10745.016,E2 -10745.016} C_VEL
LIN {X 0,Y 404.15,Z 163.133,A -85,B 0,C 180,E1 -10748.757,E2 -10748.757} C_VEL
LIN {X 0,Y 404.121,Z 163.136,A -85,B 0,C 180,E1 -10751.599,E2 -10751.599} C_VEL
LIN {X 0,Y 404.143,Z 163.137,A -85,B 0,C 180,E1 -10754.521,E2 -10754.521} C_VEL
LIN {X 0,Y 404.134,Z 163.123,A -85,B 0,C 180,E1 -10757.295,E2 -10757.295} C_VEL
LIN {X 0,Y 404.167,Z 163.14,A -85,B 0,C 180,E1 -10759.955,E2 -10759.955} C_VEL
LIN {X 0,Y 404.134,Z 163.132,A -85,B 0,C 180,E1 -10763.125,E2 -10763.125} C_VEL
LIN {X 0,Y 404.141,Z 163.121,A -85,B 0,C 180,E1 -10766.187,E2 -10766.187} C_VEL
LIN {X 0,Y 404.142,Z 163.144,A -85,B 0,C 180,E1 -10769.714,E2 -10769.714} C_VEL
LIN {X 0,Y 404.19,Z 163.128,A -85,B 0,C 180,E1 -10773.122,E2 -10773.122} C_VEL
LIN {X 0,Y 404.169,Z 163.139,A -85,B 0,C 180,E1 -10775.334,E2 -10775.334} C_VEL
LIN {X 0,Y 404.133,Z 163.136,A -85,B 0,C 180,E1 -10778.58,E2 -10778.58} C_VEL
LIN {X 0,Y 404.204,Z 163.137,A -85,B 0,C 180,E1 -10781.762,E2 -10781.762} C_VEL
LIN {X 0,Y 404.2,Z 163.123,A -85,B 0,C 180,E1 -10784.882,E2 -10784.882} C_VEL
LIN {X 0,Y 404.25,Z 163.128,A -85,B 0,C 180,E1 -10787.958,E2 -10787.958} C_VEL
LIN {X 0,Y 404.428,Z 163.103,A -85,B 0,C 180,E1 -10792.1,E2 -10792.1} C_VEL
LIN {X 0,Y 404.413,Z 163.108,A -85,B 0,C 180,E1 -10794.015,E2 -10794.015} C_VEL
LIN {X 0,Y 404.472,Z 163.093,A -85,B 0,C 180,E1 -10798.008,E2 -10798.008} C_VEL
LIN {X 0,Y 404.602,Z 163.085,A -85,B 0,C 180,E1 -10800,E2 -10800} C_VEL
LIN {X 0,Y 404.407,Z 163.107,A -85,B 0,C 180,E1 -10802.988,E2 -10802.988} C_VEL
LIN {X 0,Y 404.405,Z 163.106,A -85,B 0,C 180,E1 -10805.985,E2 -10805.985} C_VEL
LIN {X 0,Y 404.259,Z 163.128,A -85,B 0,C 180,E1 -10809.002,E2 -10809.002} C_VEL
LIN {X 0,Y 404.249,Z 163.121,A -85,B 0,C 180,E1 -10812.042,E2 -10812.042} C_VEL
LIN {X 0,Y 404.199,Z 163.138,A -85,B 0,C 180,E1 -10815.118,E2 -10815.118} C_VEL
LIN {X 0,Y 404.198,Z 163.125,A -85,B 0,C 180,E1 -10818.239,E2 -10818.239} C_VEL
LIN {X 0,Y 404.132,Z 163.145,A -85,B 0,C 180,E1 -10821.42,E2 -10821.42} C_VEL
LIN {X 0,Y 404.165,Z 163.131,A -85,B 0,C 180,E1 -10824.666,E2 -10824.666} C_VEL
LIN {X 0,Y 404.191,Z 163.132,A -85,B 0,C 180,E1 -10828,E2 -10828} C_VEL
LIN {X 0,Y 404.135,Z 163.144,A -85,B 0,C 180,E1 -10831.558,E2 -10831.558} C_VEL
LIN {X 0,Y 404.179,Z 163.121,A -85,B 0,C 180,E1 -10835.017,E2 -10835.017} C_VEL
LIN {X 0,Y 404.147,Z 163.132,A -85,B 0,C 180,E1 -10838.758,E2 -10838.758} C_VEL
LIN {X 0,Y 404.116,Z 163.143,A -85,B 0,C 180,E1 -10841.599,E2 -10841.599} C_VEL
LIN {X 0,Y 404.142,Z 163.141,A -85,B 0,C 180,E1 -10844.522,E2 -10844.522} C_VEL
LIN {X 0,Y 404.122,Z 163.143,A -85,B 0,C 180,E1 -10847.294,E2 -10847.294} C_VEL
LIN {X 0,Y 404.131,Z 163.14,A -85,B 0,C 180,E1 -10849.951,E2 -10849.951} C_VEL
LIN {X 0,Y 404.133,Z 163.142,A -85,B 0,C 180,E1 -10853.126,E2 -10853.126} C_VEL
LIN {X 0,Y 404.145,Z 163.133,A -85,B 0,C 180,E1 -10856.188,E2 -10856.188} C_VEL
LIN {X 0,Y 404.144,Z 163.137,A -85,B 0,C 180,E1 -10859.715,E2 -10859.715} C_VEL
LIN {X 0,Y 404.204,Z 163.277,A -85,B 0,C 180,E1 -10863.194,E2 -10863.194} C_VEL
LIN {X 0,Y 406.483,Z 174.778,A -85,B 0,C 180,E1 -10866.023,E2 -10866.023} C_VEL
LIN {X 0,Y 407.078,Z 179.57,A -85,B 0,C 180,E1 -10867.142,E2 -10867.142} C_VEL
LIN {X 0,Y 406.043,Z 193.964,A -85,B 0,C 180,E1 -10870.242,E2 -10870.242} C_VEL
LIN {X 0,Y 408.872,Z 209.861,A -85,B 0,C 180,E1 -10870.707,E2 -10870.707} C_VEL
LIN {X 0,Y 410.412,Z 219.887,A -85,B 0,C 180,E1 -10870.964,E2 -10870.964} C_VEL
LIN {X 0,Y 409.457,Z 301.675,A -85,B 0,C 180,E1 -10872.423,E2 -10872.423} C_VEL
LIN {X 0,Y 408.861,Z 314.896,A -85,B 0,C 180,E1 -10872.848,E2 -10872.848} C_VEL
LIN {X 0,Y 408.255,Z 327.026,A -85,B 0,C 180,E1 -10873.434,E2 -10873.434} C_VEL
LIN {X 0,Y 407.474,Z 339.263,A -85,B 0,C 180,E1 -10874.237,E2 -10874.237} C_VEL
LIN {X 0,Y 406.652,Z 350.54,A -85,B 0,C 180,E1 -10875.202,E2 -10875.202} C_VEL
LIN {X 0,Y 405.829,Z 361.249,A -85,B 0,C 180,E1 -10876.352,E2 -10876.352} C_VEL
LIN {X 0,Y 405.141,Z 369.762,A -85,B 0,C 180,E1 -10877.476,E2 -10877.476} C_VEL
LIN {X 0,Y 404.44,Z 377.614,A -85,B 0,C 180,E1 -10878.726,E2 -10878.726} C_VEL
LIN {X 0,Y 403.837,Z 385.281,A -85,B 0,C 180,E1 -10880.231,E2 -10880.231} C_VEL
LIN {X 0,Y 403.32,Z 392.349,A -85,B 0,C 180,E1 -10881.986,E2 -10881.986} C_VEL
LIN {X 0,Y 403.056,Z 397.54,A -85,B 0,C 180,E1 -10883.668,E2 -10883.668} C_VEL
LIN {X 0,Y 402.973,Z 400.641,A -85,B 0,C 180,E1 -10884.997,E2 -10884.997} C_VEL
LIN {X 0,Y 402.859,Z 402.491,A -85,B 0,C 180,E1 -10885.998,E2 -10885.998} C_VEL
LIN {X 0,Y 402.824,Z 404.87,A -85,B 0,C 180,E1 -10888,E2 -10888} C_VEL
LIN {X 0,Y 402.845,Z 405.475,A -85,B 0,C 180,E1 -10889,E2 -10889} C_VEL
LIN {X 0,Y 402.832,Z 405.689,A -85,B 0,C 180,E1 -10890,E2 -10890} C_VEL
LIN {X 0,Y 402.845,Z 405.472,A -85,B 0,C 180,E1 -10890.999,E2 -10890.999} C_VEL
LIN {X 0,Y 402.824,Z 404.867,A -85,B 0,C 180,E1 -10891.999,E2 -10891.999} C_VEL
LIN {X 0,Y 402.859,Z 402.485,A -85,B 0,C 180,E1 -10894.001,E2 -10894.001} C_VEL
LIN {X 0,Y 402.986,Z 399.561,A -85,B 0,C 180,E1 -10895.504,E2 -10895.504} C_VEL
LIN {X 0,Y 403.186,Z 395.603,A -85,B 0,C 180,E1 -10897.008,E2 -10897.008} C_VEL
LIN {X 0,Y 403.521,Z 389.514,A -85,B 0,C 180,E1 -10898.765,E2 -10898.765} C_VEL
LIN {X 0,Y 404.012,Z 382.859,A -85,B 0,C 180,E1 -10900.27,E2 -10900.27} C_VEL
LIN {X 0,Y 404.672,Z 374.6,A -85,B 0,C 180,E1 -10901.774,E2 -10901.774} C_VEL
LIN {X 0,Y 405.46,Z 366.132,A -85,B 0,C 180,E1 -10903.022,E2 -10903.022} C_VEL
LIN {X 0,Y 406.215,Z 355.847,A -85,B 0,C 180,E1 -10904.252,E2 -10904.252} C_VEL
LIN {X 0,Y 406.991,Z 345.304,A -85,B 0,C 180,E1 -10905.268,E2 -10905.268} C_VEL
LIN {X 0,Y 407.779,Z 333.942,A -85,B 0,C 180,E1 -10906.135,E2 -10906.135} C_VEL
LIN {X 0,Y 408.523,Z 322.273,A -85,B 0,C 180,E1 -10906.811,E2 -10906.811} C_VEL
LIN {X 0,Y 409.116,Z 308.818,A -85,B 0,C 180,E1 -10907.365,E2 -10907.365} C_VEL
LIN {X 0,Y 409.535,Z 295.472,A -85,B 0,C 180,E1 -10907.701,E2 -10907.701} C_VEL
LIN {X 0,Y 410.419,Z 219.12,A -85,B 0,C 180,E1 -10909.04,E2 -10909.04} C_VEL
LIN {X 0,Y 406.059,Z 194.277,A -85,B 0,C 180,E1 -10909.723,E2 -10909.723} C_VEL
LIN {X 0,Y 406.073,Z 192.629,A -85,B 0,C 180,E1 -10909.986,E2 -10909.986} C_VEL
LIN {X 0,Y 407.058,Z 179.527,A -85,B 0,C 180,E1 -10912.858,E2 -10912.858} C_VEL
LIN {X 0,Y 406.462,Z 174.501,A -85,B 0,C 180,E1 -10914.03,E2 -10914.03} C_VEL
LIN {X 0,Y 404.201,Z 163.262,A -85,B 0,C 180,E1 -10916.806,E2 -10916.806} C_VEL
LIN {X 0,Y 404.141,Z 163.137,A -85,B 0,C 180,E1 -10920.284,E2 -10920.284} C_VEL
LIN {X 0,Y 404.141,Z 163.134,A -85,B 0,C 180,E1 -10923.811,E2 -10923.811} C_VEL
LIN {X 0,Y 404.13,Z 163.141,A -85,B 0,C 180,E1 -10926.873,E2 -10926.873} C_VEL
LIN {X 0,Y 404.142,Z 163.139,A -85,B 0,C 180,E1 -10930.079,E2 -10930.079} C_VEL
LIN {X 0,Y 404.144,Z 163.14,A -85,B 0,C 180,E1 -10933.082,E2 -10933.082} C_VEL
LIN {X 0,Y 404.142,Z 163.138,A -85,B 0,C 180,E1 -10935.925,E2 -10935.925} C_VEL
LIN {X 0,Y 404.111,Z 163.146,A -85,B 0,C 180,E1 -10938.634,E2 -10938.634} C_VEL
LIN {X 0,Y 404.142,Z 163.129,A -85,B 0,C 180,E1 -10941.492,E2 -10941.492} C_VEL
LIN {X 0,Y 404.175,Z 163.122,A -85,B 0,C 180,E1 -10944.983,E2 -10944.983} C_VEL
LIN {X 0,Y 404.132,Z 163.145,A -85,B 0,C 180,E1 -10948.553,E2 -10948.553} C_VEL
LIN {X 0,Y 404.185,Z 163.133,A -85,B 0,C 180,E1 -10952,E2 -10952} C_VEL
LIN {X 0,Y 404.16,Z 163.131,A -85,B 0,C 180,E1 -10955.333,E2 -10955.333} C_VEL
LIN {X 0,Y 404.127,Z 163.145,A -85,B 0,C 180,E1 -10958.58,E2 -10958.58} C_VEL
LIN {X 0,Y 404.193,Z 163.125,A -85,B 0,C 180,E1 -10961.761,E2 -10961.761} C_VEL
LIN {X 0,Y 404.195,Z 163.138,A -85,B 0,C 180,E1 -10964.882,E2 -10964.882} C_VEL
LIN {X 0,Y 404.259,Z 163.119,A -85,B 0,C 180,E1 -10967.959,E2 -10967.959} C_VEL
LIN {X 0,Y 404.393,Z 163.111,A -85,B 0,C 180,E1 -10972.129,E2 -10972.129} C_VEL
LIN {X 0,Y 404.407,Z 163.105,A -85,B 0,C 180,E1 -10974.015,E2 -10974.015} C_VEL
LIN {X 0,Y 404.468,Z 163.099,A -85,B 0,C 180,E1 -10978.009,E2 -10978.009} C_VEL
LIN {X 0,Y 404.598,Z 163.085,A -85,B 0,C 180,E1 -10980,E2 -10980} C_VEL
LIN {X 0,Y 404.402,Z 163.103,A -85,B 0,C 180,E1 -10982.989,E2 -10982.989} C_VEL
LIN {X 0,Y 404.397,Z 163.106,A -85,B 0,C 180,E1 -10986.988,E2 -10986.988} C_VEL
LIN {X 0,Y 404.247,Z 163.117,A -85,B 0,C 180,E1 -10990.012,E2 -10990.012} C_VEL
LIN {X 0,Y 404.255,Z 163.125,A -85,B 0,C 180,E1 -10993.212,E2 -10993.212} C_VEL
LIN {X 0,Y 404.205,Z 163.129,A -85,B 0,C 180,E1 -10997.008,E2 -10997.008} C_VEL
LIN {X 0,Y 404.153,Z 163.139,A -85,B 0,C 180,E1 -11000.352,E2 -11000.352} C_VEL
LIN {X 0,Y 404.16,Z 163.135,A -85,B 0,C 180,E1 -11003.575,E2 -11003.575} C_VEL
LIN {X 0,Y 404.174,Z 163.139,A -85,B 0,C 180,E1 -11005.767,E2 -11005.767} C_VEL
LIN {X 0,Y 404.186,Z 163.131,A -85,B 0,C 180,E1 -11008.001,E2 -11008.001} C_VEL
LIN {X 0,Y 404.13,Z 163.143,A -85,B 0,C 180,E1 -11011.559,E2 -11011.559} C_VEL
LIN {X 0,Y 404.177,Z 163.107,A -85,B 0,C 180,E1 -11015.017,E2 -11015.017} C_VEL
LIN {X 0,Y 404.147,Z 163.14,A -85,B 0,C 180,E1 -11018.758,E2 -11018.758} C_VEL
LIN {X 0,Y 404.116,Z 163.141,A -85,B 0,C 180,E1 -11021.601,E2 -11021.601} C_VEL
LIN {X 0,Y 404.139,Z 163.132,A -85,B 0,C 180,E1 -11024.523,E2 -11024.523} C_VEL
LIN {X 0,Y 404.131,Z 163.144,A -85,B 0,C 180,E1 -11027.297,E2 -11027.297} C_VEL
LIN {X 0,Y 404.165,Z 163.124,A -85,B 0,C 180,E1 -11029.957,E2 -11029.957} C_VEL
LIN {X 0,Y 404.132,Z 163.144,A -85,B 0,C 180,E1 -11033.126,E2 -11033.126} C_VEL
LIN {X 0,Y 404.142,Z 163.14,A -85,B 0,C 180,E1 -11036.189,E2 -11036.189} C_VEL
LIN {X 0,Y 404.143,Z 163.14,A -85,B 0,C 180,E1 -11039.716,E2 -11039.716} C_VEL
LIN {X 0,Y 404.194,Z 163.137,A -85,B 0,C 180,E1 -11043.124,E2 -11043.124} C_VEL
LIN {X 0,Y 404.196,Z 163.224,A -85,B 0,C 180,E1 -11044.602,E2 -11044.602} C_VEL
LIN {X 0,Y 406.338,Z 174.145,A -85,B 0,C 180,E1 -11047.379,E2 -11047.379} C_VEL
LIN {X 0,Y 406.795,Z 177.544,A -85,B 0,C 180,E1 -11048.196,E2 -11048.196} C_VEL
LIN {X 0,Y 406.149,Z 187.124,A -85,B 0,C 180,E1 -11050.304,E2 -11050.304} C_VEL
LIN {X 0,Y 409.149,Z 202.827,A -85,B 0,C 180,E1 -11050.776,E2 -11050.776} C_VEL
LIN {X 0,Y 410.473,Z 210.573,A -85,B 0,C 180,E1 -11050.981,E2 -11050.981} C_VEL
LIN {X 0,Y 409.448,Z 294.939,A -85,B 0,C 180,E1 -11052.488,E2 -11052.488} C_VEL
LIN {X 0,Y 408.998,Z 308.01,A -85,B 0,C 180,E1 -11052.92,E2 -11052.92} C_VEL
LIN {X 0,Y 408.356,Z 320.06,A -85,B 0,C 180,E1 -11053.503,E2 -11053.503} C_VEL
LIN {X 0,Y 407.628,Z 331.432,A -85,B 0,C 180,E1 -11054.244,E2 -11054.244} C_VEL
LIN {X 0,Y 406.875,Z 342.411,A -85,B 0,C 180,E1 -11055.171,E2 -11055.171} C_VEL
LIN {X 0,Y 406.118,Z 353.592,A -85,B 0,C 180,E1 -11056.363,E2 -11056.363} C_VEL
LIN {X 0,Y 405.359,Z 362.16,A -85,B 0,C 180,E1 -11057.484,E2 -11057.484} C_VEL
LIN {X 0,Y 404.664,Z 370.053,A -85,B 0,C 180,E1 -11058.734,E2 -11058.734} C_VEL
LIN {X 0,Y 404.035,Z 377.771,A -85,B 0,C 180,E1 -11060.236,E2 -11060.236} C_VEL
LIN {X 0,Y 403.463,Z 384.855,A -85,B 0,C 180,E1 -11061.99,E2 -11061.99} C_VEL
LIN {X 0,Y 403.217,Z 389.491,A -85,B 0,C 180,E1 -11063.465,E2 -11063.465} C_VEL
LIN {X 0,Y 403.045,Z 393.19,A -85,B 0,C 180,E1 -11064.999,E2 -11064.999} C_VEL
LIN {X 0,Y 402.904,Z 395.059,A -85,B 0,C 180,E1 -11066,E2 -11066} C_VEL
LIN {X 0,Y 402.853,Z 396.466,A -85,B 0,C 180,E1 -11067,E2 -11067} C_VEL
LIN {X 0,Y 402.847,Z 397.701,A -85,B 0,C 180,E1 -11068.381,E2 -11068.381} C_VEL
LIN {X 0,Y 402.157,Z 398.189,A -85,B 0,C 180,E1 -11069.214,E2 -11069.214} C_VEL
LIN {X 0,Y 399.273,Z 398.276,A -85,B 0,C 180,E1 -11070.57,E2 -11070.57} C_VEL
LIN {X 0,Y 396.85,Z 397.873,A -85,B 0,C 180,E1 -11071.665,E2 -11071.665} C_VEL
LIN {X 0,Y 395.765,Z 397.081,A -85,B 0,C 180,E1 -11072.65,E2 -11072.65} C_VEL
LIN {X 0,Y 395.746,Z 396.886,A -85,B 0,C 180,E1 -11072.792,E2 -11072.792} C_VEL
LIN {X 0,Y 395.825,Z 395.274,A -85,B 0,C 180,E1 -11074.073,E2 -11074.073} C_VEL
LIN {X 0,Y 396.02,Z 392.395,A -85,B 0,C 180,E1 -11075.602,E2 -11075.602} C_VEL
LIN {X 0,Y 396.225,Z 388.494,A -85,B 0,C 180,E1 -11077.133,E2 -11077.133} C_VEL
LIN {X 0,Y 396.554,Z 383.461,A -85,B 0,C 180,E1 -11078.664,E2 -11078.664} C_VEL
LIN {X 0,Y 397.089,Z 377.128,A -85,B 0,C 180,E1 -11080.195,E2 -11080.195} C_VEL
LIN {X 0,Y 397.755,Z 369.202,A -85,B 0,C 180,E1 -11081.724,E2 -11081.724} C_VEL
LIN {X 0,Y 398.706,Z 359.344,A -85,B 0,C 180,E1 -11083.247,E2 -11083.247} C_VEL
LIN {X 0,Y 399.466,Z 349.895,A -85,B 0,C 180,E1 -11084.42,E2 -11084.42} C_VEL
LIN {X 0,Y 400.27,Z 338.763,A -85,B 0,C 180,E1 -11085.531,E2 -11085.531} C_VEL
LIN {X 0,Y 401.16,Z 327.56,A -85,B 0,C 180,E1 -11086.409,E2 -11086.409} C_VEL
LIN {X 0,Y 401.818,Z 316.198,A -85,B 0,C 180,E1 -11087.101,E2 -11087.101} C_VEL
LIN {X 0,Y 402.453,Z 303.237,A -85,B 0,C 180,E1 -11087.663,E2 -11087.663} C_VEL
LIN {X 0,Y 402.853,Z 289.374,A -85,B 0,C 180,E1 -11088.039,E2 -11088.039} C_VEL
LIN {X 0,Y 403.645,Z 210.372,A -85,B 0,C 180,E1 -11089.459,E2 -11089.459} C_VEL
LIN {X 0,Y 399.283,Z 187.299,A -85,B 0,C 180,E1 -11090.141,E2 -11090.141} C_VEL
LIN {X 0,Y 399.334,Z 184.95,A -85,B 0,C 180,E1 -11090.609,E2 -11090.609} C_VEL
LIN {X 0,Y 399.818,Z 178.031,A -85,B 0,C 180,E1 -11092.205,E2 -11092.205} C_VEL
LIN {X 0,Y 397.664,Z 166.543,A -85,B 0,C 180,E1 -11095.097,E2 -11095.097} C_VEL
LIN {X 0,Y 397.147,Z 164.037,A -85,B 0,C 180,E1 -11095.834,E2 -11095.834} C_VEL
LIN {X 0,Y 397.123,Z 164.014,A -85,B 0,C 180,E1 -11098.543,E2 -11098.543} C_VEL
LIN {X 0,Y 397.079,Z 164.018,A -85,B 0,C 180,E1 -11102.071,E2 -11102.071} C_VEL
LIN {X 0,Y 397.12,Z 164.007,A -85,B 0,C 180,E1 -11105.503,E2 -11105.503} C_VEL
LIN {X 0,Y 397.126,Z 164.007,A -85,B 0,C 180,E1 -11108.86,E2 -11108.86} C_VEL
LIN {X 0,Y 397.067,Z 164.022,A -85,B 0,C 180,E1 -11112.267,E2 -11112.267} C_VEL
LIN {X 0,Y 397.085,Z 164.014,A -85,B 0,C 180,E1 -11115.068,E2 -11115.068} C_VEL
LIN {X 0,Y 397.064,Z 164.01,A -85,B 0,C 180,E1 -11118.021,E2 -11118.021} C_VEL
LIN {X 0,Y 397.129,Z 164.014,A -85,B 0,C 180,E1 -11121.138,E2 -11121.138} C_VEL
LIN {X 0,Y 397.116,Z 163.985,A -85,B 0,C 180,E1 -11124.496,E2 -11124.496} C_VEL
LIN {X 0,Y 397.075,Z 164.017,A -85,B 0,C 180,E1 -11127.928,E2 -11127.928} C_VEL
LIN {X 0,Y 397.118,Z 164.016,A -85,B 0,C 180,E1 -11131.456,E2 -11131.456} C_VEL
LIN {X 0,Y 397.148,Z 164.013,A -85,B 0,C 180,E1 -11134.487,E2 -11134.487} C_VEL
LIN {X 0,Y 397.09,Z 164.013,A -85,B 0,C 180,E1 -11138.181,E2 -11138.181} C_VEL
LIN {X 0,Y 397.157,Z 164.014,A -85,B 0,C 180,E1 -11141.426,E2 -11141.426} C_VEL
LIN {X 0,Y 397.173,Z 163.998,A -85,B 0,C 180,E1 -11144.608,E2 -11144.608} C_VEL
LIN {X 0,Y 397.213,Z 164.007,A -85,B 0,C 180,E1 -11147.742,E2 -11147.742} C_VEL
LIN {X 0,Y 397.389,Z 163.98,A -85,B 0,C 180,E1 -11152.041,E2 -11152.041} C_VEL
LIN {X 0,Y 397.244,Z 163.999,A -85,B 0,C 180,E1 -11154.925,E2 -11154.925} C_VEL
LIN {X 0,Y 397.441,Z 163.968,A -85,B 0,C 180,E1 -11157.973,E2 -11157.973} C_VEL
LIN {X 0,Y 397.571,Z 163.96,A -85,B 0,C 180,E1 -11160,E2 -11160} C_VEL
LIN {X 0,Y 397.367,Z 163.985,A -85,B 0,C 180,E1 -11163.041,E2 -11163.041} C_VEL
LIN {X 0,Y 397.356,Z 163.983,A -85,B 0,C 180,E1 -11166.092,E2 -11166.092} C_VEL
LIN {X 0,Y 397.229,Z 164.005,A -85,B 0,C 180,E1 -11169.162,E2 -11169.162} C_VEL
LIN {X 0,Y 397.213,Z 163.997,A -85,B 0,C 180,E1 -11172.258,E2 -11172.258} C_VEL
LIN {X 0,Y 397.173,Z 164.012,A -85,B 0,C 180,E1 -11175.392,E2 -11175.392} C_VEL
LIN {X 0,Y 397.152,Z 164.003,A -85,B 0,C 180,E1 -11178.574,E2 -11178.574} C_VEL
LIN {X 0,Y 397.09,Z 164.018,A -85,B 0,C 180,E1 -11181.819,E2 -11181.819} C_VEL
LIN {X 0,Y 397.148,Z 164.015,A -85,B 0,C 180,E1 -11185.513,E2 -11185.513} C_VEL
LIN {X 0,Y 397.118,Z 164.014,A -85,B 0,C 180,E1 -11188.544,E2 -11188.544} C_VEL
LIN {X 0,Y 397.074,Z 164.022,A -85,B 0,C 180,E1 -11192.072,E2 -11192.072} C_VEL
LIN {X 0,Y 397.115,Z 163.994,A -85,B 0,C 180,E1 -11195.504,E2 -11195.504} C_VEL
LIN {X 0,Y 397.123,Z 164.008,A -85,B 0,C 180,E1 -11198.861,E2 -11198.861} C_VEL
LIN {X 0,Y 397.061,Z 164.021,A -85,B 0,C 180,E1 -11202.268,E2 -11202.268} C_VEL
LIN {X 0,Y 397.084,Z 164.025,A -85,B 0,C 180,E1 -11205.069,E2 -11205.069} C_VEL
LIN {X 0,Y 397.052,Z 164.023,A -85,B 0,C 180,E1 -11208.024,E2 -11208.024} C_VEL
LIN {X 0,Y 397.093,Z 164.005,A -85,B 0,C 180,E1 -11211.146,E2 -11211.146} C_VEL
LIN {X 0,Y 397.118,Z 164.021,A -85,B 0,C 180,E1 -11214.497,E2 -11214.497} C_VEL
LIN {X 0,Y 397.078,Z 164.024,A -85,B 0,C 180,E1 -11217.929,E2 -11217.929} C_VEL
LIN {X 0,Y 397.118,Z 164.017,A -85,B 0,C 180,E1 -11220.296,E2 -11220.296} C_VEL
LIN {X 0,Y 397.155,Z 164.135,A -85,B 0,C 180,E1 -11222.892,E2 -11222.892} C_VEL
LIN {X 0,Y 399.281,Z 174.73,A -85,B 0,C 180,E1 -11225.567,E2 -11225.567} C_VEL
LIN {X 0,Y 400.138,Z 180.697,A -85,B 0,C 180,E1 -11226.996,E2 -11226.996} C_VEL
LIN {X 0,Y 399.139,Z 193.902,A -85,B 0,C 180,E1 -11229.886,E2 -11229.886} C_VEL
LIN {X 0,Y 402.158,Z 210.55,A -85,B 0,C 180,E1 -11230.386,E2 -11230.386} C_VEL
LIN {X 0,Y 403.724,Z 221.54,A -85,B 0,C 180,E1 -11230.668,E2 -11230.668} C_VEL
LIN {X 0,Y 402.688,Z 301.622,A -85,B 0,C 180,E1 -11232.118,E2 -11232.118} C_VEL
LIN {X 0,Y 402.098,Z 314.84,A -85,B 0,C 180,E1 -11232.551,E2 -11232.551} C_VEL
LIN {X 0,Y 401.445,Z 326.967,A -85,B 0,C 180,E1 -11233.145,E2 -11233.145} C_VEL
LIN {X 0,Y 400.622,Z 339.202,A -85,B 0,C 180,E1 -11233.961,E2 -11233.961} C_VEL
LIN {X 0,Y 399.744,Z 350.697,A -85,B 0,C 180,E1 -11234.962,E2 -11234.962} C_VEL
LIN {X 0,Y 398.896,Z 361.186,A -85,B 0,C 180,E1 -11236.11,E2 -11236.11} C_VEL
LIN {X 0,Y 398.187,Z 369.699,A -85,B 0,C 180,E1 -11237.254,E2 -11237.254} C_VEL
LIN {X 0,Y 397.462,Z 377.551,A -85,B 0,C 180,E1 -11238.526,E2 -11238.526} C_VEL
LIN {X 0,Y 396.823,Z 385.218,A -85,B 0,C 180,E1 -11240.056,E2 -11240.056} C_VEL
LIN {X 0,Y 396.263,Z 392.285,A -85,B 0,C 180,E1 -11241.843,E2 -11241.843} C_VEL
LIN {X 0,Y 395.985,Z 397.128,A -85,B 0,C 180,E1 -11243.426,E2 -11243.426} C_VEL
LIN {X 0,Y 395.89,Z 400.576,A -85,B 0,C 180,E1 -11244.907,E2 -11244.907} C_VEL
LIN {X 0,Y 395.784,Z 402.427,A -85,B 0,C 180,E1 -11245.927,E2 -11245.927} C_VEL
LIN {X 0,Y 395.722,Z 404.805,A -85,B 0,C 180,E1 -11247.964,E2 -11247.964} C_VEL
LIN {X 0,Y 395.756,Z 405.41,A -85,B 0,C 180,E1 -11248.982,E2 -11248.982} C_VEL
LIN {X 0,Y 395.76,Z 405.624,A -85,B 0,C 180,E1 -11250,E2 -11250} C_VEL
LIN {X 0,Y 395.756,Z 405.407,A -85,B 0,C 180,E1 -11251.017,E2 -11251.017} C_VEL
LIN {X 0,Y 395.7,Z 403.809,A -85,B 0,C 180,E1 -11253.054,E2 -11253.054} C_VEL
LIN {X 0,Y 395.783,Z 402.419,A -85,B 0,C 180,E1 -11254.073,E2 -11254.073} C_VEL
LIN {X 0,Y 395.888,Z 399.495,A -85,B 0,C 180,E1 -11255.603,E2 -11255.603} C_VEL
LIN {X 0,Y 396.101,Z 395.537,A -85,B 0,C 180,E1 -11257.134,E2 -11257.134} C_VEL
LIN {X 0,Y 396.467,Z 389.447,A -85,B 0,C 180,E1 -11258.922,E2 -11258.922} C_VEL
LIN {X 0,Y 397.02,Z 382.792,A -85,B 0,C 180,E1 -11260.453,E2 -11260.453} C_VEL
LIN {X 0,Y 397.712,Z 374.533,A -85,B 0,C 180,E1 -11261.983,E2 -11261.983} C_VEL
LIN {X 0,Y 398.515,Z 366.064,A -85,B 0,C 180,E1 -11263.253,E2 -11263.253} C_VEL
LIN {X 0,Y 399.26,Z 356.567,A -85,B 0,C 180,E1 -11264.419,E2 -11264.419} C_VEL
LIN {X 0,Y 400.12,Z 345.235,A -85,B 0,C 180,E1 -11265.536,E2 -11265.536} C_VEL
LIN {X 0,Y 400.951,Z 333.872,A -85,B 0,C 180,E1 -11266.417,E2 -11266.417} C_VEL
LIN {X 0,Y 401.731,Z 322.201,A -85,B 0,C 180,E1 -11267.104,E2 -11267.104} C_VEL
LIN {X 0,Y 402.34,Z 308.743,A -85,B 0,C 180,E1 -11267.667,E2 -11267.667} C_VEL
LIN {X 0,Y 402.794,Z 295.388,A -85,B 0,C 180,E1 -11268.008,E2 -11268.008} C_VEL
LIN {X 0,Y 403.585,Z 219.266,A -85,B 0,C 180,E1 -11269.371,E2 -11269.371} C_VEL
LIN {X 0,Y 399.158,Z 194.205,A -85,B 0,C 180,E1 -11270.079,E2 -11270.079} C_VEL
LIN {X 0,Y 399.163,Z 192.561,A -85,B 0,C 180,E1 -11270.348,E2 -11270.348} C_VEL
LIN {X 0,Y 400.113,Z 180.651,A -85,B 0,C 180,E1 -11273.005,E2 -11273.005} C_VEL
LIN {X 0,Y 399.278,Z 174.682,A -85,B 0,C 180,E1 -11274.432,E2 -11274.432} C_VEL
LIN {X 0,Y 397.152,Z 164.118,A -85,B 0,C 180,E1 -11277.107,E2 -11277.107} C_VEL
LIN {X 0,Y 397.097,Z 164.017,A -85,B 0,C 180,E1 -11279.862,E2 -11279.862} C_VEL
LIN {X 0,Y 397.115,Z 164.009,A -85,B 0,C 180,E1 -11283.717,E2 -11283.717} C_VEL
LIN {X 0,Y 397.086,Z 164.013,A -85,B 0,C 180,E1 -11287.207,E2 -11287.207} C_VEL
LIN {X 0,Y 397.071,Z 164.02,A -85,B 0,C 180,E1 -11290.44,E2 -11290.44} C_VEL
LIN {X 0,Y 397.094,Z 164.02,A -85,B 0,C 180,E1 -11293.648,E2 -11293.648} C_VEL
LIN {X 0,Y 397.095,Z 164.016,A -85,B 0,C 180,E1 -11296.52,E2 -11296.52} C_VEL
LIN {X 0,Y 397.105,Z 164.017,A -85,B 0,C 180,E1 -11300.422,E2 -11300.422} C_VEL
LIN {X 0,Y 397.099,Z 163.996,A -85,B 0,C 180,E1 -11304.264,E2 -11304.264} C_VEL
LIN {X 0,Y 397.106,Z 164.016,A -85,B 0,C 180,E1 -11306.726,E2 -11306.726} C_VEL
LIN {X 0,Y 397.115,Z 164.012,A -85,B 0,C 180,E1 -11310.295,E2 -11310.295} C_VEL
LIN {X 0,Y 397.184,Z 164.009,A -85,B 0,C 180,E1 -11312.609,E2 -11312.609} C_VEL
LIN {X 0,Y 397.115,Z 164.007,A -85,B 0,C 180,E1 -11315.981,E2 -11315.981} C_VEL
LIN {X 0,Y 397.128,Z 164.013,A -85,B 0,C 180,E1 -11319.704,E2 -11319.704} C_VEL
LIN {X 0,Y 397.171,Z 164.004,A -85,B 0,C 180,E1 -11322.845,E2 -11322.845} C_VEL
LIN {X 0,Y 397.217,Z 164.003,A -85,B 0,C 180,E1 -11326.702,E2 -11326.702} C_VEL
LIN {X 0,Y 397.211,Z 163.998,A -85,B 0,C 180,E1 -11329.809,E2 -11329.809} C_VEL
LIN {X 0,Y 397.339,Z 163.988,A -85,B 0,C 180,E1 -11332.888,E2 -11332.888} C_VEL
LIN {X 0,Y 397.239,Z 163.99,A -85,B 0,C 180,E1 -11334.925,E2 -11334.925} C_VEL
LIN {X 0,Y 397.437,Z 163.975,A -85,B 0,C 180,E1 -11337.973,E2 -11337.973} C_VEL
LIN {X 0,Y 397.568,Z 163.961,A -85,B 0,C 180,E1 -11340,E2 -11340} C_VEL
LIN {X 0,Y 397.361,Z 163.979,A -85,B 0,C 180,E1 -11343.042,E2 -11343.042} C_VEL
LIN {X 0,Y 397.35,Z 163.983,A -85,B 0,C 180,E1 -11347.112,E2 -11347.112} C_VEL
LIN {X 0,Y 397.206,Z 163.996,A -85,B 0,C 180,E1 -11350.191,E2 -11350.191} C_VEL
LIN {X 0,Y 397.216,Z 164.002,A -85,B 0,C 180,E1 -11353.322,E2 -11353.322} C_VEL
LIN {X 0,Y 397.171,Z 164.005,A -85,B 0,C 180,E1 -11357.156,E2 -11357.156} C_VEL
LIN {X 0,Y 397.092,Z 164.014,A -85,B 0,C 180,E1 -11360.731,E2 -11360.731} C_VEL
LIN {X 0,Y 397.123,Z 164.015,A -85,B 0,C 180,E1 -11364.019,E2 -11364.019} C_VEL
LIN {X 0,Y 397.185,Z 164.001,A -85,B 0,C 180,E1 -11367.391,E2 -11367.391} C_VEL
LIN {X 0,Y 397.069,Z 164.022,A -85,B 0,C 180,E1 -11370.883,E2 -11370.883} C_VEL
LIN {X 0,Y 397.117,Z 163.988,A -85,B 0,C 180,E1 -11374.494,E2 -11374.494} C_VEL
LIN {X 0,Y 397.095,Z 164.019,A -85,B 0,C 180,E1 -11378.276,E2 -11378.276} C_VEL
LIN {X 0,Y 397.082,Z 164.018,A -85,B 0,C 180,E1 -11380.91,E2 -11380.91} C_VEL
LIN {X 0,Y 397.094,Z 164,A -85,B 0,C 180,E1 -11383.65,E2 -11383.65} C_VEL
LIN {X 0,Y 397.097,Z 164.02,A -85,B 0,C 180,E1 -11386.522,E2 -11386.522} C_VEL
LIN {X 0,Y 397.108,Z 164.003,A -85,B 0,C 180,E1 -11390.424,E2 -11390.424} C_VEL
LIN {X 0,Y 397.105,Z 164.011,A -85,B 0,C 180,E1 -11394.267,E2 -11394.267} C_VEL
LIN {X 0,Y 397.112,Z 164.018,A -85,B 0,C 180,E1 -11396.728,E2 -11396.728} C_VEL
LIN {X 0,Y 397.123,Z 164.019,A -85,B 0,C 180,E1 -11400.297,E2 -11400.297} C_VEL
LIN {X 0,Y 397.193,Z 164.011,A -85,B 0,C 180,E1 -11402.611,E2 -11402.611} C_VEL
LIN {X 0,Y 397.188,Z 164.226,A -85,B 0,C 180,E1 -11404.384,E2 -11404.384} C_VEL
LIN {X 0,Y 399.365,Z 175.308,A -85,B 0,C 180,E1 -11407.223,E2 -11407.223} C_VEL
LIN {X 0,Y 399.864,Z 178.757,A -85,B 0,C 180,E1 -11408.07,E2 -11408.07} C_VEL
LIN {X 0,Y 399.234,Z 187.196,A -85,B 0,C 180,E1 -11409.949,E2 -11409.949} C_VEL
LIN {X 0,Y 402.736,Z 205.19,A -85,B 0,C 180,E1 -11410.499,E2 -11410.499} C_VEL
LIN {X 0,Y 403.732,Z 211.333,A -85,B 0,C 180,E1 -11410.663,E2 -11410.663} C_VEL
LIN {X 0,Y 402.682,Z 295.02,A -85,B 0,C 180,E1 -11412.184,E2 -11412.184} C_VEL
LIN {X 0,Y 402.218,Z 308.086,A -85,B 0,C 180,E1 -11412.622,E2 -11412.622} C_VEL
LIN {X 0,Y 401.472,Z 321.237,A -85,B 0,C 180,E1 -11413.278,E2 -11413.278} C_VEL
LIN {X 0,Y 400.703,Z 333.092,A -85,B 0,C 180,E1 -11414.095,E2 -11414.095} C_VEL
LIN {X 0,Y 399.897,Z 344.3,A -85,B 0,C 180,E1 -11415.09,E2 -11415.09} C_VEL
LIN {X 0,Y 399.131,Z 354.723,A -85,B 0,C 180,E1 -11416.249,E2 -11416.249} C_VEL
LIN {X 0,Y 398.254,Z 363.927,A -85,B 0,C 180,E1 -11417.516,E2 -11417.516} C_VEL
LIN {X 0,Y 397.472,Z 372.867,A -85,B 0,C 180,E1 -11419.043,E2 -11419.043} C_VEL
LIN {X 0,Y 396.853,Z 380.065,A -85,B 0,C 180,E1 -11420.572,E2 -11420.572} C_VEL
LIN {X 0,Y 396.424,Z 384.922,A -85,B 0,C 180,E1 -11421.847,E2 -11421.847} C_VEL
LIN {X 0,Y 396.136,Z 389.907,A -85,B 0,C 180,E1 -11423.474,E2 -11423.474} C_VEL
LIN {X 0,Y 395.967,Z 393.256,A -85,B 0,C 180,E1 -11424.909,E2 -11424.909} C_VEL
LIN {X 0,Y 395.828,Z 395.124,A -85,B 0,C 180,E1 -11425.928,E2 -11425.928} C_VEL
LIN {X 0,Y 395.756,Z 396.532,A -85,B 0,C 180,E1 -11426.947,E2 -11426.947} C_VEL
LIN {X 0,Y 395.75,Z 397.781,A -85,B 0,C 180,E1 -11428.377,E2 -11428.377} C_VEL
LIN {X 0,Y 395.76,Z 398.382,A -85,B 0,C 180,E1 -11430,E2 -11430} C_VEL
LIN {X 0,Y 395.76,Z 398.193,A -85,B 0,C 180,E1 -11431.018,E2 -11431.018} C_VEL
LIN {X 0,Y 395.746,Z 396.886,A -85,B 0,C 180,E1 -11432.792,E2 -11432.792} C_VEL
LIN {X 0,Y 395.115,Z 395.948,A -85,B 0,C 180,E1 -11433.632,E2 -11433.632} C_VEL
LIN {X 0,Y 392.372,Z 393.818,A -85,B 0,C 180,E1 -11434.985,E2 -11434.985} C_VEL
LIN {X 0,Y 390.09,Z 391.605,A -85,B 0,C 180,E1 -11436.058,E2 -11436.058} C_VEL
LIN {X 0,Y 389.175,Z 389.631,A -85,B 0,C 180,E1 -11436.871,E2 -11436.871} C_VEL
LIN {X 0,Y 389.135,Z 388.886,A -85,B 0,C 180,E1 -11437.143,E2 -11437.143} C_VEL
LIN {X 0,Y 389.528,Z 383.525,A -85,B 0,C 180,E1 -11438.822,E2 -11438.822} C_VEL
LIN {X 0,Y 390.077,Z 377.191,A -85,B 0,C 180,E1 -11440.38,E2 -11440.38} C_VEL
LIN {X 0,Y 390.804,Z 369.264,A -85,B 0,C 180,E1 -11441.936,E2 -11441.936} C_VEL
LIN {X 0,Y 391.787,Z 359.406,A -85,B 0,C 180,E1 -11443.486,E2 -11443.486} C_VEL
LIN {X 0,Y 392.541,Z 349.878,A -85,B 0,C 180,E1 -11444.689,E2 -11444.689} C_VEL
LIN {X 0,Y 393.425,Z 338.823,A -85,B 0,C 180,E1 -11445.808,E2 -11445.808} C_VEL
LIN {X 0,Y 394.337,Z 327.619,A -85,B 0,C 180,E1 -11446.701,E2 -11446.701} C_VEL
LIN {X 0,Y 395.041,Z 316.254,A -85,B 0,C 180,E1 -11447.404,E2 -11447.404} C_VEL
LIN {X 0,Y 395.719,Z 303.288,A -85,B 0,C 180,E1 -11447.974,E2 -11447.974} C_VEL
LIN {X 0,Y 396.076,Z 290.922,A -85,B 0,C 180,E1 -11448.325,E2 -11448.325} C_VEL
LIN {X 0,Y 397.042,Z 211.839,A -85,B 0,C 180,E1 -11449.769,E2 -11449.769} C_VEL
LIN {X 0,Y 392.404,Z 187.354,A -85,B 0,C 180,E1 -11450.51,E2 -11450.51} C_VEL
LIN {X 0,Y 392.633,Z 183.701,A -85,B 0,C 180,E1 -11451.289,E2 -11451.289} C_VEL
LIN {X 0,Y 392.856,Z 179.24,A -85,B 0,C 180,E1 -11452.343,E2 -11452.343} C_VEL
LIN {X 0,Y 390.455,Z 166.596,A -85,B 0,C 180,E1 -11455.594,E2 -11455.594} C_VEL
LIN {X 0,Y 390.115,Z 164.908,A -85,B 0,C 180,E1 -11456.138,E2 -11456.138} C_VEL
LIN {X 0,Y 390.06,Z 164.896,A -85,B 0,C 180,E1 -11459.109,E2 -11459.109} C_VEL
LIN {X 0,Y 390.043,Z 164.901,A -85,B 0,C 180,E1 -11462.721,E2 -11462.721} C_VEL
LIN {X 0,Y 390.056,Z 164.888,A -85,B 0,C 180,E1 -11465.825,E2 -11465.825} C_VEL
LIN {X 0,Y 390.067,Z 164.884,A -85,B 0,C 180,E1 -11469.217,E2 -11469.217} C_VEL
LIN {X 0,Y 390.041,Z 164.899,A -85,B 0,C 180,E1 -11472.374,E2 -11472.374} C_VEL
LIN {X 0,Y 390.042,Z 164.891,A -85,B 0,C 180,E1 -11475.354,E2 -11475.354} C_VEL
LIN {X 0,Y 390.029,Z 164.888,A -85,B 0,C 180,E1 -11478.186,E2 -11478.186} C_VEL
LIN {X 0,Y 390.089,Z 164.891,A -85,B 0,C 180,E1 -11480.907,E2 -11480.907} C_VEL
LIN {X 0,Y 390.082,Z 164.859,A -85,B 0,C 180,E1 -11484.793,E2 -11484.793} C_VEL
LIN {X 0,Y 390.02,Z 164.901,A -85,B 0,C 180,E1 -11488.495,E2 -11488.495} C_VEL
LIN {X 0,Y 390.114,Z 164.883,A -85,B 0,C 180,E1 -11492.07,E2 -11492.07} C_VEL
LIN {X 0,Y 390.073,Z 164.896,A -85,B 0,C 180,E1 -11495.519,E2 -11495.519} C_VEL
LIN {X 0,Y 390.083,Z 164.889,A -85,B 0,C 180,E1 -11499.53,E2 -11499.53} C_VEL
LIN {X 0,Y 390.133,Z 164.884,A -85,B 0,C 180,E1 -11503.248,E2 -11503.248} C_VEL
LIN {X 0,Y 390.189,Z 164.877,A -85,B 0,C 180,E1 -11506.561,E2 -11506.561} C_VEL
LIN {X 0,Y 390.199,Z 164.864,A -85,B 0,C 180,E1 -11510.671,E2 -11510.671} C_VEL
LIN {X 0,Y 390.311,Z 164.859,A -85,B 0,C 180,E1 -11512.759,E2 -11512.759} C_VEL
LIN {X 0,Y 390.216,Z 164.874,A -85,B 0,C 180,E1 -11514.833,E2 -11514.833} C_VEL
LIN {X 0,Y 390.41,Z 164.843,A -85,B 0,C 180,E1 -11517.937,E2 -11517.937} C_VEL
LIN {X 0,Y 390.541,Z 164.836,A -85,B 0,C 180,E1 -11520,E2 -11520} C_VEL
LIN {X 0,Y 390.301,Z 164.865,A -85,B 0,C 180,E1 -11523.097,E2 -11523.097} C_VEL
LIN {X 0,Y 390.309,Z 164.861,A -85,B 0,C 180,E1 -11526.202,E2 -11526.202} C_VEL
LIN {X 0,Y 390.187,Z 164.88,A -85,B 0,C 180,E1 -11529.329,E2 -11529.329} C_VEL
LIN {X 0,Y 390.165,Z 164.875,A -85,B 0,C 180,E1 -11532.483,E2 -11532.483} C_VEL
LIN {X 0,Y 390.133,Z 164.885,A -85,B 0,C 180,E1 -11535.677,E2 -11535.677} C_VEL
LIN {X 0,Y 390.096,Z 164.884,A -85,B 0,C 180,E1 -11538.923,E2 -11538.923} C_VEL
LIN {X 0,Y 390.032,Z 164.896,A -85,B 0,C 180,E1 -11542.235,E2 -11542.235} C_VEL
LIN {X 0,Y 390.114,Z 164.889,A -85,B 0,C 180,E1 -11545.744,E2 -11545.744} C_VEL
LIN {X 0,Y 390.054,Z 164.892,A -85,B 0,C 180,E1 -11549.11,E2 -11549.11} C_VEL
LIN {X 0,Y 390.039,Z 164.901,A -85,B 0,C 180,E1 -11552.722,E2 -11552.722} C_VEL
LIN {X 0,Y 390.052,Z 164.872,A -85,B 0,C 180,E1 -11555.825,E2 -11555.825} C_VEL
LIN {X 0,Y 390.064,Z 164.892,A -85,B 0,C 180,E1 -11559.218,E2 -11559.218} C_VEL
LIN {X 0,Y 390.036,Z 164.897,A -85,B 0,C 180,E1 -11562.374,E2 -11562.374} C_VEL
LIN {X 0,Y 390.041,Z 164.899,A -85,B 0,C 180,E1 -11565.355,E2 -11565.355} C_VEL
LIN {X 0,Y 390.016,Z 164.9,A -85,B 0,C 180,E1 -11568.185,E2 -11568.185} C_VEL
LIN {X 0,Y 390.057,Z 164.883,A -85,B 0,C 180,E1 -11570.904,E2 -11570.904} C_VEL
LIN {X 0,Y 390.084,Z 164.893,A -85,B 0,C 180,E1 -11574.793,E2 -11574.793} C_VEL
LIN {X 0,Y 390.023,Z 164.901,A -85,B 0,C 180,E1 -11578.496,E2 -11578.496} C_VEL
LIN {X 0,Y 390.038,Z 164.881,A -85,B 0,C 180,E1 -11582.064,E2 -11582.064} C_VEL
LIN {X 0,Y 390.116,Z 165.165,A -85,B 0,C 180,E1 -11582.653,E2 -11582.653} C_VEL
LIN {X 0,Y 392.296,Z 175.855,A -85,B 0,C 180,E1 -11585.385,E2 -11585.385} C_VEL
LIN {X 0,Y 393.204,Z 181.824,A -85,B 0,C 180,E1 -11586.845,E2 -11586.845} C_VEL
LIN {X 0,Y 392.243,Z 193.816,A -85,B 0,C 180,E1 -11589.514,E2 -11589.514} C_VEL
LIN {X 0,Y 394.795,Z 207.518,A -85,B 0,C 180,E1 -11589.948,E2 -11589.948} C_VEL
LIN {X 0,Y 397.018,Z 221.405,A -85,B 0,C 180,E1 -11590.326,E2 -11590.326} C_VEL
LIN {X 0,Y 395.936,Z 301.57,A -85,B 0,C 180,E1 -11591.802,E2 -11591.802} C_VEL
LIN {X 0,Y 395.334,Z 314.783,A -85,B 0,C 180,E1 -11592.242,E2 -11592.242} C_VEL
LIN {X 0,Y 394.647,Z 326.908,A -85,B 0,C 180,E1 -11592.845,E2 -11592.845} C_VEL
LIN {X 0,Y 393.783,Z 339.142,A -85,B 0,C 180,E1 -11593.674,E2 -11593.674} C_VEL
LIN {X 0,Y 392.839,Z 350.969,A -85,B 0,C 180,E1 -11594.726,E2 -11594.726} C_VEL
LIN {X 0,Y 391.914,Z 362.164,A -85,B 0,C 180,E1 -11595.99,E2 -11595.99} C_VEL
LIN {X 0,Y 391.098,Z 371.308,A -85,B 0,C 180,E1 -11597.283,E2 -11597.283} C_VEL
LIN {X 0,Y 390.223,Z 380.217,A -85,B 0,C 180,E1 -11598.836,E2 -11598.836} C_VEL
LIN {X 0,Y 389.586,Z 387.384,A -85,B 0,C 180,E1 -11600.394,E2 -11600.394} C_VEL
LIN {X 0,Y 389.222,Z 392.221,A -85,B 0,C 180,E1 -11601.694,E2 -11601.694} C_VEL
LIN {X 0,Y 388.913,Z 397.064,A -85,B 0,C 180,E1 -11603.306,E2 -11603.306} C_VEL
LIN {X 0,Y 388.806,Z 400.512,A -85,B 0,C 180,E1 -11604.814,E2 -11604.814} C_VEL
LIN {X 0,Y 388.71,Z 402.363,A -85,B 0,C 180,E1 -11605.852,E2 -11605.852} C_VEL
LIN {X 0,Y 388.619,Z 404.741,A -85,B 0,C 180,E1 -11607.927,E2 -11607.927} C_VEL
LIN {X 0,Y 388.655,Z 405.345,A -85,B 0,C 180,E1 -11608.963,E2 -11608.963} C_VEL
LIN {X 0,Y 388.672,Z 405.559,A -85,B 0,C 180,E1 -11610,E2 -11610} C_VEL
LIN {X 0,Y 388.655,Z 405.342,A -85,B 0,C 180,E1 -11611.036,E2 -11611.036} C_VEL
LIN {X 0,Y 388.61,Z 403.744,A -85,B 0,C 180,E1 -11613.11,E2 -11613.11} C_VEL
LIN {X 0,Y 388.71,Z 402.354,A -85,B 0,C 180,E1 -11614.147,E2 -11614.147} C_VEL
LIN {X 0,Y 388.808,Z 399.059,A -85,B 0,C 180,E1 -11615.869,E2 -11615.869} C_VEL
LIN {X 0,Y 389.031,Z 395.471,A -85,B 0,C 180,E1 -11617.264,E2 -11617.264} C_VEL
LIN {X 0,Y 389.437,Z 389.381,A -85,B 0,C 180,E1 -11619.085,E2 -11619.085} C_VEL
LIN {X 0,Y 390.031,Z 382.726,A -85,B 0,C 180,E1 -11620.643,E2 -11620.643} C_VEL
LIN {X 0,Y 390.757,Z 374.466,A -85,B 0,C 180,E1 -11622.2,E2 -11622.2} C_VEL
LIN {X 0,Y 391.582,Z 365.997,A -85,B 0,C 180,E1 -11623.492,E2 -11623.492} C_VEL
LIN {X 0,Y 392.409,Z 356.025,A -85,B 0,C 180,E1 -11624.729,E2 -11624.729} C_VEL
LIN {X 0,Y 393.271,Z 345.166,A -85,B 0,C 180,E1 -11625.814,E2 -11625.814} C_VEL
LIN {X 0,Y 394.15,Z 333.802,A -85,B 0,C 180,E1 -11626.709,E2 -11626.709} C_VEL
LIN {X 0,Y 394.959,Z 322.129,A -85,B 0,C 180,E1 -11627.407,E2 -11627.407} C_VEL
LIN {X 0,Y 395.596,Z 308.668,A -85,B 0,C 180,E1 -11627.979,E2 -11627.979} C_VEL
LIN {X 0,Y 396.066,Z 295.304,A -85,B 0,C 180,E1 -11628.324,E2 -11628.324} C_VEL
LIN {X 0,Y 396.914,Z 220.338,A -85,B 0,C 180,E1 -11629.688,E2 -11629.688} C_VEL
LIN {X 0,Y 392.304,Z 194.439,A -85,B 0,C 180,E1 -11630.435,E2 -11630.435} C_VEL
LIN {X 0,Y 392.254,Z 193.15,A -85,B 0,C 180,E1 -11630.585,E2 -11630.585} C_VEL
LIN {X 0,Y 393.176,Z 181.775,A -85,B 0,C 180,E1 -11633.156,E2 -11633.156} C_VEL
LIN {X 0,Y 392.066,Z 174.608,A -85,B 0,C 180,E1 -11634.912,E2 -11634.912} C_VEL
LIN {X 0,Y 390.095,Z 164.976,A -85,B 0,C 180,E1 -11637.421,E2 -11637.421} C_VEL
LIN {X 0,Y 390.034,Z 164.894,A -85,B 0,C 180,E1 -11640.299,E2 -11640.299} C_VEL
LIN {X 0,Y 390.065,Z 164.887,A -85,B 0,C 180,E1 -11644.023,E2 -11644.023} C_VEL
LIN {X 0,Y 390.035,Z 164.886,A -85,B 0,C 180,E1 -11647.549,E2 -11647.549} C_VEL
LIN {X 0,Y 390.042,Z 164.899,A -85,B 0,C 180,E1 -11650.819,E2 -11650.819} C_VEL
LIN {X 0,Y 390.048,Z 164.897,A -85,B 0,C 180,E1 -11653.885,E2 -11653.885} C_VEL
LIN {X 0,Y 390.05,Z 164.893,A -85,B 0,C 180,E1 -11656.789,E2 -11656.789} C_VEL
LIN {X 0,Y 390.049,Z 164.897,A -85,B 0,C 180,E1 -11659.559,E2 -11659.559} C_VEL
LIN {X 0,Y 390.034,Z 164.877,A -85,B 0,C 180,E1 -11662.449,E2 -11662.449} C_VEL
LIN {X 0,Y 390.06,Z 164.889,A -85,B 0,C 180,E1 -11665.974,E2 -11665.974} C_VEL
LIN {X 0,Y 390.037,Z 164.892,A -85,B 0,C 180,E1 -11669.868,E2 -11669.868} C_VEL
LIN {X 0,Y 390.103,Z 164.892,A -85,B 0,C 180,E1 -11673.231,E2 -11673.231} C_VEL
LIN {X 0,Y 390.057,Z 164.89,A -85,B 0,C 180,E1 -11676.763,E2 -11676.763} C_VEL
LIN {X 0,Y 390.092,Z 164.89,A -85,B 0,C 180,E1 -11679.982,E2 -11679.982} C_VEL
LIN {X 0,Y 390.127,Z 164.885,A -85,B 0,C 180,E1 -11683.248,E2 -11683.248} C_VEL
LIN {X 0,Y 390.184,Z 164.881,A -85,B 0,C 180,E1 -11686.561,E2 -11686.561} C_VEL
LIN {X 0,Y 390.163,Z 164.875,A -85,B 0,C 180,E1 -11689.623,E2 -11689.623} C_VEL
LIN {X 0,Y 390.291,Z 164.867,A -85,B 0,C 180,E1 -11692.759,E2 -11692.759} C_VEL
LIN {X 0,Y 390.211,Z 164.866,A -85,B 0,C 180,E1 -11694.833,E2 -11694.833} C_VEL
LIN {X 0,Y 390.406,Z 164.851,A -85,B 0,C 180,E1 -11697.937,E2 -11697.937} C_VEL
LIN {X 0,Y 390.537,Z 164.836,A -85,B 0,C 180,E1 -11700,E2 -11700} C_VEL
LIN {X 0,Y 390.296,Z 164.859,A -85,B 0,C 180,E1 -11703.097,E2 -11703.097} C_VEL
LIN {X 0,Y 390.294,Z 164.863,A -85,B 0,C 180,E1 -11706.709,E2 -11706.709} C_VEL
LIN {X 0,Y 390.193,Z 164.864,A -85,B 0,C 180,E1 -11709.329,E2 -11709.329} C_VEL
LIN {X 0,Y 390.184,Z 164.878,A -85,B 0,C 180,E1 -11713.439,E2 -11713.439} C_VEL
LIN {X 0,Y 390.138,Z 164.881,A -85,B 0,C 180,E1 -11717.308,E2 -11717.308} C_VEL
LIN {X 0,Y 390.077,Z 164.891,A -85,B 0,C 180,E1 -11720.471,E2 -11720.471} C_VEL
LIN {X 0,Y 390.08,Z 164.888,A -85,B 0,C 180,E1 -11723.352,E2 -11723.352} C_VEL
LIN {X 0,Y 390.104,Z 164.884,A -85,B 0,C 180,E1 -11726.769,E2 -11726.769} C_VEL
LIN {X 0,Y 390.03,Z 164.903,A -85,B 0,C 180,E1 -11730.301,E2 -11730.301} C_VEL
LIN {X 0,Y 390.06,Z 164.872,A -85,B 0,C 180,E1 -11734.026,E2 -11734.026} C_VEL
LIN {X 0,Y 390.036,Z 164.889,A -85,B 0,C 180,E1 -11737.552,E2 -11737.552} C_VEL
LIN {X 0,Y 390.05,Z 164.894,A -85,B 0,C 180,E1 -11740.822,E2 -11740.822} C_VEL
LIN {X 0,Y 390.048,Z 164.878,A -85,B 0,C 180,E1 -11743.887,E2 -11743.887} C_VEL
LIN {X 0,Y 390.052,Z 164.897,A -85,B 0,C 180,E1 -11746.791,E2 -11746.791} C_VEL
LIN {X 0,Y 390.052,Z 164.882,A -85,B 0,C 180,E1 -11749.562,E2 -11749.562} C_VEL
LIN {X 0,Y 390.038,Z 164.9,A -85,B 0,C 180,E1 -11752.451,E2 -11752.451} C_VEL
LIN {X 0,Y 390.065,Z 164.889,A -85,B 0,C 180,E1 -11755.977,E2 -11755.977} C_VEL
LIN {X 0,Y 390.045,Z 164.898,A -85,B 0,C 180,E1 -11759.87,E2 -11759.87} C_VEL
LIN {X 0,Y 390.112,Z 164.89,A -85,B 0,C 180,E1 -11763.233,E2 -11763.233} C_VEL
LIN {X 0,Y 390.124,Z 165.083,A -85,B 0,C 180,E1 -11764.083,E2 -11764.083} C_VEL
LIN {X 0,Y 392.387,Z 176.518,A -85,B 0,C 180,E1 -11767.074,E2 -11767.074} C_VEL
LIN {X 0,Y 392.933,Z 179.969,A -85,B 0,C 180,E1 -11767.939,E2 -11767.939} C_VEL
LIN {X 0,Y 392.36,Z 187.214,A -85,B 0,C 180,E1 -11769.577,E2 -11769.577} C_VEL
LIN {X 0,Y 394.33,Z 197.339,A -85,B 0,C 180,E1 -11769.915,E2 -11769.915} C_VEL
LIN {X 0,Y 397,Z 211.731,A -85,B 0,C 180,E1 -11770.328,E2 -11770.328} C_VEL
LIN {X 0,Y 395.98,Z 293.92,A -85,B 0,C 180,E1 -11771.839,E2 -11771.839} C_VEL
LIN {X 0,Y 395.546,Z 306.639,A -85,B 0,C 180,E1 -11772.253,E2 -11772.253} C_VEL
LIN {X 0,Y 394.792,Z 320.206,A -85,B 0,C 180,E1 -11772.92,E2 -11772.92} C_VEL
LIN {X 0,Y 393.99,Z 331.574,A -85,B 0,C 180,E1 -11773.684,E2 -11773.684} C_VEL
LIN {X 0,Y 393.049,Z 343.704,A -85,B 0,C 180,E1 -11774.755,E2 -11774.755} C_VEL
LIN {X 0,Y 392.318,Z 353.73,A -85,B 0,C 180,E1 -11775.873,E2 -11775.873} C_VEL
LIN {X 0,Y 391.501,Z 362.296,A -85,B 0,C 180,E1 -11777.034,E2 -11777.034} C_VEL
LIN {X 0,Y 390.69,Z 370.189,A -85,B 0,C 180,E1 -11778.325,E2 -11778.325} C_VEL
LIN {X 0,Y 390.008,Z 377.905,A -85,B 0,C 180,E1 -11779.882,E2 -11779.882} C_VEL
LIN {X 0,Y 389.378,Z 384.989,A -85,B 0,C 180,E1 -11781.698,E2 -11781.698} C_VEL
LIN {X 0,Y 389.055,Z 390.321,A -85,B 0,C 180,E1 -11783.485,E2 -11783.485} C_VEL
LIN {X 0,Y 388.894,Z 393.322,A -85,B 0,C 180,E1 -11784.816,E2 -11784.816} C_VEL
LIN {X 0,Y 388.755,Z 395.19,A -85,B 0,C 180,E1 -11785.854,E2 -11785.854} C_VEL
LIN {X 0,Y 388.664,Z 396.597,A -85,B 0,C 180,E1 -11786.891,E2 -11786.891} C_VEL
LIN {X 0,Y 388.667,Z 397.597,A -85,B 0,C 180,E1 -11787.928,E2 -11787.928} C_VEL
LIN {X 0,Y 388.673,Z 398.447,A -85,B 0,C 180,E1 -11790,E2 -11790} C_VEL
LIN {X 0,Y 388.66,Z 398.258,A -85,B 0,C 180,E1 -11791.037,E2 -11791.037} C_VEL
LIN {X 0,Y 388.65,Z 396.993,A -85,B 0,C 180,E1 -11792.797,E2 -11792.797} C_VEL
LIN {X 0,Y 388.752,Z 395.338,A -85,B 0,C 180,E1 -11794.147,E2 -11794.147} C_VEL
LIN {X 0,Y 388.931,Z 392.459,A -85,B 0,C 180,E1 -11795.704,E2 -11795.704} C_VEL
LIN {X 0,Y 389.135,Z 388.886,A -85,B 0,C 180,E1 -11797.143,E2 -11797.143} C_VEL
LIN {X 0,Y 388.639,Z 386.6,A -85,B 0,C 180,E1 -11797.942,E2 -11797.942} C_VEL
LIN {X 0,Y 386.178,Z 382.45,A -85,B 0,C 180,E1 -11799.223,E2 -11799.223} C_VEL
LIN {X 0,Y 383.774,Z 377.641,A -85,B 0,C 180,E1 -11800.467,E2 -11800.467} C_VEL
LIN {X 0,Y 383.372,Z 374.32,A -85,B 0,C 180,E1 -11801.197,E2 -11801.197} C_VEL
LIN {X 0,Y 384.17,Z 366.292,A -85,B 0,C 180,E1 -11802.681,E2 -11802.681} C_VEL
LIN {X 0,Y 385.116,Z 357.547,A -85,B 0,C 180,E1 -11803.993,E2 -11803.993} C_VEL
LIN {X 0,Y 385.915,Z 346.785,A -85,B 0,C 180,E1 -11805.311,E2 -11805.311} C_VEL
LIN {X 0,Y 386.847,Z 335.981,A -85,B 0,C 180,E1 -11806.355,E2 -11806.355} C_VEL
LIN {X 0,Y 387.773,Z 323.859,A -85,B 0,C 180,E1 -11807.264,E2 -11807.264} C_VEL
LIN {X 0,Y 388.587,Z 311.164,A -85,B 0,C 180,E1 -11807.974,E2 -11807.974} C_VEL
LIN {X 0,Y 389.108,Z 298.553,A -85,B 0,C 180,E1 -11808.46,E2 -11808.46} C_VEL
LIN {X 0,Y 389.394,Z 284.238,A -85,B 0,C 180,E1 -11808.787,E2 -11808.787} C_VEL
LIN {X 0,Y 390.273,Z 212.221,A -85,B 0,C 180,E1 -11810.12,E2 -11810.12} C_VEL
LIN {X 0,Y 385.561,Z 187.666,A -85,B 0,C 180,E1 -11810.877,E2 -11810.877} C_VEL
LIN {X 0,Y 385.533,Z 186.231,A -85,B 0,C 180,E1 -11811.102,E2 -11811.102} C_VEL
LIN {X 0,Y 385.907,Z 180.453,A -85,B 0,C 180,E1 -11812.485,E2 -11812.485} C_VEL
LIN {X 0,Y 383.728,Z 168.948,A -85,B 0,C 180,E1 -11815.493,E2 -11815.493} C_VEL
LIN {X 0,Y 383.072,Z 165.801,A -85,B 0,C 180,E1 -11816.417,E2 -11816.417} C_VEL
LIN {X 0,Y 382.993,Z 165.779,A -85,B 0,C 180,E1 -11819.699,E2 -11819.699} C_VEL
LIN {X 0,Y 383.004,Z 165.776,A -85,B 0,C 180,E1 -11823.4,E2 -11823.4} C_VEL
LIN {X 0,Y 383.032,Z 165.767,A -85,B 0,C 180,E1 -11826.164,E2 -11826.164} C_VEL
LIN {X 0,Y 383.007,Z 165.757,A -85,B 0,C 180,E1 -11829.958,E2 -11829.958} C_VEL
LIN {X 0,Y 383.004,Z 165.776,A -85,B 0,C 180,E1 -11832.778,E2 -11832.778} C_VEL
LIN {X 0,Y 382.995,Z 165.76,A -85,B 0,C 180,E1 -11835.789,E2 -11835.789} C_VEL
LIN {X 0,Y 382.987,Z 165.773,A -85,B 0,C 180,E1 -11838.795,E2 -11838.795} C_VEL
LIN {X 0,Y 382.998,Z 165.77,A -85,B 0,C 180,E1 -11842.096,E2 -11842.096} C_VEL
LIN {X 0,Y 383.015,Z 165.739,A -85,B 0,C 180,E1 -11845.332,E2 -11845.332} C_VEL
LIN {X 0,Y 382.979,Z 165.776,A -85,B 0,C 180,E1 -11849.081,E2 -11849.081} C_VEL
LIN {X 0,Y 383.053,Z 165.761,A -85,B 0,C 180,E1 -11852.698,E2 -11852.698} C_VEL
LIN {X 0,Y 383.046,Z 165.769,A -85,B 0,C 180,E1 -11855.039,E2 -11855.039} C_VEL
LIN {X 0,Y 382.987,Z 165.77,A -85,B 0,C 180,E1 -11858.469,E2 -11858.469} C_VEL
LIN {X 0,Y 383.084,Z 165.766,A -85,B 0,C 180,E1 -11861.827,E2 -11861.827} C_VEL
LIN {X 0,Y 383.104,Z 165.751,A -85,B 0,C 180,E1 -11865.118,E2 -11865.118} C_VEL
LIN {X 0,Y 383.091,Z 165.761,A -85,B 0,C 180,E1 -11868.358,E2 -11868.358} C_VEL
LIN {X 0,Y 383.298,Z 165.732,A -85,B 0,C 180,E1 -11871.934,E2 -11871.934} C_VEL
LIN {X 0,Y 383.189,Z 165.75,A -85,B 0,C 180,E1 -11874.738,E2 -11874.738} C_VEL
LIN {X 0,Y 383.378,Z 165.718,A -85,B 0,C 180,E1 -11877.899,E2 -11877.899} C_VEL
LIN {X 0,Y 383.51,Z 165.712,A -85,B 0,C 180,E1 -11880,E2 -11880} C_VEL
LIN {X 0,Y 383.238,Z 165.744,A -85,B 0,C 180,E1 -11883.154,E2 -11883.154} C_VEL
LIN {X 0,Y 383.264,Z 165.738,A -85,B 0,C 180,E1 -11886.317,E2 -11886.317} C_VEL
LIN {X 0,Y 383.137,Z 165.756,A -85,B 0,C 180,E1 -11889.502,E2 -11889.502} C_VEL
LIN {X 0,Y 383.12,Z 165.762,A -85,B 0,C 180,E1 -11893.536,E2 -11893.536} C_VEL
LIN {X 0,Y 383.088,Z 165.759,A -85,B 0,C 180,E1 -11897.069,E2 -11897.069} C_VEL
LIN {X 0,Y 383.023,Z 165.772,A -85,B 0,C 180,E1 -11900.647,E2 -11900.647} C_VEL
LIN {X 0,Y 383.017,Z 165.764,A -85,B 0,C 180,E1 -11903.808,E2 -11903.808} C_VEL
LIN {X 0,Y 383.075,Z 165.765,A -85,B 0,C 180,E1 -11906.124,E2 -11906.124} C_VEL
LIN {X 0,Y 382.988,Z 165.772,A -85,B 0,C 180,E1 -11909.7,E2 -11909.7} C_VEL
LIN {X 0,Y 382.999,Z 165.771,A -85,B 0,C 180,E1 -11913.401,E2 -11913.401} C_VEL
LIN {X 0,Y 383.028,Z 165.744,A -85,B 0,C 180,E1 -11916.165,E2 -11916.165} C_VEL
LIN {X 0,Y 383.005,Z 165.773,A -85,B 0,C 180,E1 -11919.959,E2 -11919.959} C_VEL
LIN {X 0,Y 383.003,Z 165.771,A -85,B 0,C 180,E1 -11922.779,E2 -11922.779} C_VEL
LIN {X 0,Y 382.993,Z 165.775,A -85,B 0,C 180,E1 -11925.789,E2 -11925.789} C_VEL
LIN {X 0,Y 382.965,Z 165.784,A -85,B 0,C 180,E1 -11928.8,E2 -11928.8} C_VEL
LIN {X 0,Y 382.992,Z 165.761,A -85,B 0,C 180,E1 -11932.098,E2 -11932.098} C_VEL
LIN {X 0,Y 383.018,Z 165.767,A -85,B 0,C 180,E1 -11935.332,E2 -11935.332} C_VEL
LIN {X 0,Y 382.982,Z 165.772,A -85,B 0,C 180,E1 -11939.082,E2 -11939.082} C_VEL
LIN {X 0,Y 383.045,Z 165.875,A -85,B 0,C 180,E1 -11942.265,E2 -11942.265} C_VEL
LIN {X 0,Y 385.087,Z 175.787,A -85,B 0,C 180,E1 -11944.892,E2 -11944.892} C_VEL
LIN {X 0,Y 386.264,Z 182.951,A -85,B 0,C 180,E1 -11946.688,E2 -11946.688} C_VEL
LIN {X 0,Y 385.375,Z 193.817,A -85,B 0,C 180,E1 -11949.139,E2 -11949.139} C_VEL
LIN {X 0,Y 389.371,Z 215.729,A -85,B 0,C 180,E1 -11949.815,E2 -11949.815} C_VEL
LIN {X 0,Y 390.368,Z 222.43,A -85,B 0,C 180,E1 -11949.997,E2 -11949.997} C_VEL
LIN {X 0,Y 389.196,Z 301.518,A -85,B 0,C 180,E1 -11951.476,E2 -11951.476} C_VEL
LIN {X 0,Y 388.591,Z 314.727,A -85,B 0,C 180,E1 -11951.924,E2 -11951.924} C_VEL
LIN {X 0,Y 387.864,Z 326.85,A -85,B 0,C 180,E1 -11952.536,E2 -11952.536} C_VEL
LIN {X 0,Y 386.981,Z 339.081,A -85,B 0,C 180,E1 -11953.379,E2 -11953.379} C_VEL
LIN {X 0,Y 386.008,Z 350.651,A -85,B 0,C 180,E1 -11954.422,E2 -11954.422} C_VEL
LIN {X 0,Y 385.107,Z 360.831,A -85,B 0,C 180,E1 -11955.573,E2 -11955.573} C_VEL
LIN {X 0,Y 384.326,Z 369.574,A -85,B 0,C 180,E1 -11956.786,E2 -11956.786} C_VEL
LIN {X 0,Y 383.51,Z 377.425,A -85,B 0,C 180,E1 -11958.102,E2 -11958.102} C_VEL
LIN {X 0,Y 382.781,Z 385.09,A -85,B 0,C 180,E1 -11959.687,E2 -11959.687} C_VEL
LIN {X 0,Y 382.169,Z 392.157,A -85,B 0,C 180,E1 -11961.54,E2 -11961.54} C_VEL
LIN {X 0,Y 381.852,Z 396.857,A -85,B 0,C 180,E1 -11963.129,E2 -11963.129} C_VEL
LIN {X 0,Y 381.707,Z 400.447,A -85,B 0,C 180,E1 -11964.718,E2 -11964.718} C_VEL
LIN {X 0,Y 381.639,Z 402.299,A -85,B 0,C 180,E1 -11965.775,E2 -11965.775} C_VEL
LIN {X 0,Y 381.517,Z 404.676,A -85,B 0,C 180,E1 -11967.888,E2 -11967.888} C_VEL
LIN {X 0,Y 381.554,Z 405.28,A -85,B 0,C 180,E1 -11968.944,E2 -11968.944} C_VEL
LIN {X 0,Y 381.572,Z 405.494,A -85,B 0,C 180,E1 -11970,E2 -11970} C_VEL
LIN {X 0,Y 381.553,Z 405.277,A -85,B 0,C 180,E1 -11971.055,E2 -11971.055} C_VEL
LIN {X 0,Y 381.524,Z 403.679,A -85,B 0,C 180,E1 -11973.167,E2 -11973.167} C_VEL
LIN {X 0,Y 381.639,Z 402.288,A -85,B 0,C 180,E1 -11974.224,E2 -11974.224} C_VEL
LIN {X 0,Y 381.752,Z 398.452,A -85,B 0,C 180,E1 -11976.208,E2 -11976.208} C_VEL
LIN {X 0,Y 382.055,Z 393.816,A -85,B 0,C 180,E1 -11977.929,E2 -11977.929} C_VEL
LIN {X 0,Y 382.482,Z 388.305,A -85,B 0,C 180,E1 -11979.518,E2 -11979.518} C_VEL
LIN {X 0,Y 383.117,Z 381.425,A -85,B 0,C 180,E1 -11981.105,E2 -11981.105} C_VEL
LIN {X 0,Y 383.978,Z 372.815,A -85,B 0,C 180,E1 -11982.687,E2 -11982.687} C_VEL
LIN {X 0,Y 384.856,Z 364.126,A -85,B 0,C 180,E1 -11983.982,E2 -11983.982} C_VEL
LIN {X 0,Y 385.724,Z 353.579,A -85,B 0,C 180,E1 -11985.264,E2 -11985.264} C_VEL
LIN {X 0,Y 386.681,Z 342.128,A -85,B 0,C 180,E1 -11986.362,E2 -11986.362} C_VEL
LIN {X 0,Y 387.643,Z 329.816,A -85,B 0,C 180,E1 -11987.269,E2 -11987.269} C_VEL
LIN {X 0,Y 388.428,Z 318.154,A -85,B 0,C 180,E1 -11987.913,E2 -11987.913} C_VEL
LIN {X 0,Y 388.994,Z 305.718,A -85,B 0,C 180,E1 -11988.397,E2 -11988.397} C_VEL
LIN {X 0,Y 389.379,Z 289.852,A -85,B 0,C 180,E1 -11988.753,E2 -11988.753} C_VEL
LIN {X 0,Y 390.263,Z 221.238,A -85,B 0,C 180,E1 -11990.019,E2 -11990.019} C_VEL
LIN {X 0,Y 385.418,Z 194.122,A -85,B 0,C 180,E1 -11990.824,E2 -11990.824} C_VEL
LIN {X 0,Y 385.401,Z 193.077,A -85,B 0,C 180,E1 -11990.969,E2 -11990.969} C_VEL
LIN {X 0,Y 386.231,Z 182.898,A -85,B 0,C 180,E1 -11993.313,E2 -11993.313} C_VEL
LIN {X 0,Y 385.06,Z 175.732,A -85,B 0,C 180,E1 -11995.108,E2 -11995.108} C_VEL
LIN {X 0,Y 383.042,Z 165.854,A -85,B 0,C 180,E1 -11997.734,E2 -11997.734} C_VEL
LIN {X 0,Y 382.979,Z 165.773,A -85,B 0,C 180,E1 -12000.918,E2 -12000.918} C_VEL
LIN {X 0,Y 383.014,Z 165.768,A -85,B 0,C 180,E1 -12004.667,E2 -12004.667} C_VEL
LIN {X 0,Y 382.99,Z 165.761,A -85,B 0,C 180,E1 -12007.902,E2 -12007.902} C_VEL
LIN {X 0,Y 382.972,Z 165.781,A -85,B 0,C 180,E1 -12011.347,E2 -12011.347} C_VEL
LIN {X 0,Y 382.989,Z 165.776,A -85,B 0,C 180,E1 -12014.302,E2 -12014.302} C_VEL
LIN {X 0,Y 383.004,Z 165.771,A -85,B 0,C 180,E1 -12017.239,E2 -12017.239} C_VEL
LIN {X 0,Y 383.006,Z 165.774,A -85,B 0,C 180,E1 -12020.413,E2 -12020.413} C_VEL
LIN {X 0,Y 383.016,Z 165.748,A -85,B 0,C 180,E1 -12024.043,E2 -12024.043} C_VEL
LIN {X 0,Y 382.977,Z 165.778,A -85,B 0,C 180,E1 -12027.577,E2 -12027.577} C_VEL
LIN {X 0,Y 382.982,Z 165.772,A -85,B 0,C 180,E1 -12030.299,E2 -12030.299} C_VEL
LIN {X 0,Y 383.07,Z 165.765,A -85,B 0,C 180,E1 -12034.02,E2 -12034.02} C_VEL
LIN {X 0,Y 382.98,Z 165.777,A -85,B 0,C 180,E1 -12037.333,E2 -12037.333} C_VEL
LIN {X 0,Y 383.047,Z 165.766,A -85,B 0,C 180,E1 -12040.716,E2 -12040.716} C_VEL
LIN {X 0,Y 383.069,Z 165.763,A -85,B 0,C 180,E1 -12044.026,E2 -12044.026} C_VEL
LIN {X 0,Y 383.13,Z 165.751,A -85,B 0,C 180,E1 -12047.284,E2 -12047.284} C_VEL
LIN {X 0,Y 383.142,Z 165.755,A -85,B 0,C 180,E1 -12050.498,E2 -12050.498} C_VEL
LIN {X 0,Y 383.268,Z 165.737,A -85,B 0,C 180,E1 -12053.683,E2 -12053.683} C_VEL
LIN {X 0,Y 383.373,Z 165.727,A -85,B 0,C 180,E1 -12057.899,E2 -12057.899} C_VEL
LIN {X 0,Y 383.507,Z 165.712,A -85,B 0,C 180,E1 -12060,E2 -12060} C_VEL
LIN {X 0,Y 383.232,Z 165.738,A -85,B 0,C 180,E1 -12063.154,E2 -12063.154} C_VEL
LIN {X 0,Y 383.253,Z 165.742,A -85,B 0,C 180,E1 -12066.705,E2 -12066.705} C_VEL
LIN {X 0,Y 383.249,Z 165.734,A -85,B 0,C 180,E1 -12068.436,E2 -12068.436} C_VEL
LIN {X 0,Y 383.085,Z 165.761,A -85,B 0,C 180,E1 -12071.643,E2 -12071.643} C_VEL
LIN {X 0,Y 383.099,Z 165.753,A -85,B 0,C 180,E1 -12074.882,E2 -12074.882} C_VEL
LIN {X 0,Y 383.079,Z 165.766,A -85,B 0,C 180,E1 -12078.173,E2 -12078.173} C_VEL
LIN {X 0,Y 382.983,Z 165.77,A -85,B 0,C 180,E1 -12081.532,E2 -12081.532} C_VEL
LIN {X 0,Y 383.043,Z 165.769,A -85,B 0,C 180,E1 -12084.961,E2 -12084.961} C_VEL
LIN {X 0,Y 383.031,Z 165.768,A -85,B 0,C 180,E1 -12088.494,E2 -12088.494} C_VEL
LIN {X 0,Y 383.001,Z 165.77,A -85,B 0,C 180,E1 -12092.151,E2 -12092.151} C_VEL
LIN {X 0,Y 383.01,Z 165.742,A -85,B 0,C 180,E1 -12094.669,E2 -12094.669} C_VEL
LIN {X 0,Y 382.992,Z 165.769,A -85,B 0,C 180,E1 -12097.905,E2 -12097.905} C_VEL
LIN {X 0,Y 382.977,Z 165.775,A -85,B 0,C 180,E1 -12101.349,E2 -12101.349} C_VEL
LIN {X 0,Y 382.989,Z 165.76,A -85,B 0,C 180,E1 -12104.304,E2 -12104.304} C_VEL
LIN {X 0,Y 383.005,Z 165.775,A -85,B 0,C 180,E1 -12107.241,E2 -12107.241} C_VEL
LIN {X 0,Y 383.009,Z 165.758,A -85,B 0,C 180,E1 -12110.415,E2 -12110.415} C_VEL
LIN {X 0,Y 383.022,Z 165.768,A -85,B 0,C 180,E1 -12114.046,E2 -12114.046} C_VEL
LIN {X 0,Y 382.984,Z 165.78,A -85,B 0,C 180,E1 -12117.579,E2 -12117.579} C_VEL
LIN {X 0,Y 382.991,Z 165.78,A -85,B 0,C 180,E1 -12120.301,E2 -12120.301} C_VEL
LIN {X 0,Y 383.07,Z 165.866,A -85,B 0,C 180,E1 -12123.731,E2 -12123.731} C_VEL
LIN {X 0,Y 385.217,Z 176.582,A -85,B 0,C 180,E1 -12126.622,E2 -12126.622} C_VEL
LIN {X 0,Y 385.916,Z 181.998,A -85,B 0,C 180,E1 -12127.997,E2 -12127.997} C_VEL
LIN {X 0,Y 385.512,Z 187.286,A -85,B 0,C 180,E1 -12129.198,E2 -12129.198} C_VEL
LIN {X 0,Y 387.986,Z 199.98,A -85,B 0,C 180,E1 -12129.621,E2 -12129.621} C_VEL
LIN {X 0,Y 390.344,Z 212.804,A -85,B 0,C 180,E1 -12129.997,E2 -12129.997} C_VEL
LIN {X 0,Y 389.261,Z 294.004,A -85,B 0,C 180,E1 -12131.514,E2 -12131.514} C_VEL
LIN {X 0,Y 388.786,Z 306.715,A -85,B 0,C 180,E1 -12131.934,E2 -12131.934} C_VEL
LIN {X 0,Y 388.025,Z 320.279,A -85,B 0,C 180,E1 -12132.612,E2 -12132.612} C_VEL
LIN {X 0,Y 387.192,Z 331.645,A -85,B 0,C 180,E1 -12133.389,E2 -12133.389} C_VEL
LIN {X 0,Y 386.273,Z 342.966,A -85,B 0,C 180,E1 -12134.397,E2 -12134.397} C_VEL
LIN {X 0,Y 385.432,Z 353.799,A -85,B 0,C 180,E1 -12135.616,E2 -12135.616} C_VEL
LIN {X 0,Y 384.582,Z 362.364,A -85,B 0,C 180,E1 -12136.796,E2 -12136.796} C_VEL
LIN {X 0,Y 383.728,Z 370.257,A -85,B 0,C 180,E1 -12138.11,E2 -12138.11} C_VEL
LIN {X 0,Y 383.007,Z 377.973,A -85,B 0,C 180,E1 -12139.695,E2 -12139.695} C_VEL
LIN {X 0,Y 382.332,Z 385.056,A -85,B 0,C 180,E1 -12141.544,E2 -12141.544} C_VEL
LIN {X 0,Y 382.01,Z 389.776,A -85,B 0,C 180,E1 -12143.133,E2 -12143.133} C_VEL
LIN {X 0,Y 381.82,Z 393.388,A -85,B 0,C 180,E1 -12144.72,E2 -12144.72} C_VEL
LIN {X 0,Y 381.685,Z 395.256,A -85,B 0,C 180,E1 -12145.777,E2 -12145.777} C_VEL
LIN {X 0,Y 381.575,Z 396.662,A -85,B 0,C 180,E1 -12146.833,E2 -12146.833} C_VEL
LIN {X 0,Y 381.566,Z 397.662,A -85,B 0,C 180,E1 -12147.889,E2 -12147.889} C_VEL
LIN {X 0,Y 381.573,Z 398.512,A -85,B 0,C 180,E1 -12150,E2 -12150} C_VEL
LIN {X 0,Y 381.56,Z 398.323,A -85,B 0,C 180,E1 -12151.056,E2 -12151.056} C_VEL
LIN {X 0,Y 381.566,Z 397.735,A -85,B 0,C 180,E1 -12152.112,E2 -12152.112} C_VEL
LIN {X 0,Y 381.681,Z 395.402,A -85,B 0,C 180,E1 -12154.224,E2 -12154.224} C_VEL
LIN {X 0,Y 381.873,Z 392.002,A -85,B 0,C 180,E1 -12156.05,E2 -12156.05} C_VEL
LIN {X 0,Y 382.213,Z 387.059,A -85,B 0,C 180,E1 -12157.927,E2 -12157.927} C_VEL
LIN {X 0,Y 382.788,Z 380.6,A -85,B 0,C 180,E1 -12159.778,E2 -12159.778} C_VEL
LIN {X 0,Y 383.372,Z 374.32,A -85,B 0,C 180,E1 -12161.197,E2 -12161.197} C_VEL
LIN {X 0,Y 383.024,Z 370.827,A -85,B 0,C 180,E1 -12161.909,E2 -12161.909} C_VEL
LIN {X 0,Y 380.896,Z 364.862,A -85,B 0,C 180,E1 -12163.054,E2 -12163.054} C_VEL
LIN {X 0,Y 378.818,Z 358.354,A -85,B 0,C 180,E1 -12164.136,E2 -12164.136} C_VEL
LIN {X 0,Y 378.542,Z 353.995,A -85,B 0,C 180,E1 -12164.738,E2 -12164.738} C_VEL
LIN {X 0,Y 379.302,Z 344.338,A -85,B 0,C 180,E1 -12165.861,E2 -12165.861} C_VEL
LIN {X 0,Y 380.332,Z 332.88,A -85,B 0,C 180,E1 -12166.92,E2 -12166.92} C_VEL
LIN {X 0,Y 381.24,Z 320.884,A -85,B 0,C 180,E1 -12167.778,E2 -12167.778} C_VEL
LIN {X 0,Y 381.954,Z 308.268,A -85,B 0,C 180,E1 -12168.436,E2 -12168.436} C_VEL
LIN {X 0,Y 382.605,Z 295.181,A -85,B 0,C 180,E1 -12168.89,E2 -12168.89} C_VEL
LIN {X 0,Y 383.204,Z 254.7,A -85,B 0,C 180,E1 -12169.678,E2 -12169.678} C_VEL
LIN {X 0,Y 383.655,Z 213.472,A -85,B 0,C 180,E1 -12170.459,E2 -12170.459} C_VEL
LIN {X 0,Y 378.823,Z 188.538,A -85,B 0,C 180,E1 -12171.235,E2 -12171.235} C_VEL
LIN {X 0,Y 378.687,Z 186.913,A -85,B 0,C 180,E1 -12171.371,E2 -12171.371} C_VEL
LIN {X 0,Y 378.936,Z 181.659,A -85,B 0,C 180,E1 -12172.636,E2 -12172.636} C_VEL
LIN {X 0,Y 376.643,Z 169.657,A -85,B 0,C 180,E1 -12175.839,E2 -12175.839} C_VEL
LIN {X 0,Y 376.049,Z 166.661,A -85,B 0,C 180,E1 -12176.762,E2 -12176.762} C_VEL
LIN {X 0,Y 375.957,Z 166.647,A -85,B 0,C 180,E1 -12180.693,E2 -12180.693} C_VEL
LIN {X 0,Y 375.96,Z 166.645,A -85,B 0,C 180,E1 -12184.111,E2 -12184.111} C_VEL
LIN {X 0,Y 375.953,Z 166.655,A -85,B 0,C 180,E1 -12186.741,E2 -12186.741} C_VEL
LIN {X 0,Y 375.987,Z 166.631,A -85,B 0,C 180,E1 -12189.97,E2 -12189.97} C_VEL
LIN {X 0,Y 375.929,Z 166.659,A -85,B 0,C 180,E1 -12193.765,E2 -12193.765} C_VEL
LIN {X 0,Y 375.932,Z 166.632,A -85,B 0,C 180,E1 -12196.81,E2 -12196.81} C_VEL
LIN {X 0,Y 375.961,Z 166.653,A -85,B 0,C 180,E1 -12200.537,E2 -12200.537} C_VEL
LIN {X 0,Y 375.961,Z 166.632,A -85,B 0,C 180,E1 -12203.495,E2 -12203.495} C_VEL
LIN {X 0,Y 375.957,Z 166.622,A -85,B 0,C 180,E1 -12205.888,E2 -12205.888} C_VEL
LIN {X 0,Y 375.961,Z 166.654,A -85,B 0,C 180,E1 -12209.687,E2 -12209.687} C_VEL
LIN {X 0,Y 376.016,Z 166.639,A -85,B 0,C 180,E1 -12213.347,E2 -12213.347} C_VEL
LIN {X 0,Y 375.974,Z 166.645,A -85,B 0,C 180,E1 -12216.887,E2 -12216.887} C_VEL
LIN {X 0,Y 375.993,Z 166.648,A -85,B 0,C 180,E1 -12220.339,E2 -12220.339} C_VEL
LIN {X 0,Y 376.023,Z 166.635,A -85,B 0,C 180,E1 -12223.718,E2 -12223.718} C_VEL
LIN {X 0,Y 376.098,Z 166.633,A -85,B 0,C 180,E1 -12227.042,E2 -12227.042} C_VEL
LIN {X 0,Y 376.113,Z 166.619,A -85,B 0,C 180,E1 -12230.318,E2 -12230.318} C_VEL
LIN {X 0,Y 376.223,Z 166.614,A -85,B 0,C 180,E1 -12232.486,E2 -12232.486} C_VEL
LIN {X 0,Y 376.162,Z 166.625,A -85,B 0,C 180,E1 -12234.64,E2 -12234.64} C_VEL
LIN {X 0,Y 376.344,Z 166.594,A -85,B 0,C 180,E1 -12237.86,E2 -12237.86} C_VEL
LIN {X 0,Y 376.48,Z 166.588,A -85,B 0,C 180,E1 -12240,E2 -12240} C_VEL
LIN {X 0,Y 376.176,Z 166.622,A -85,B 0,C 180,E1 -12243.213,E2 -12243.213} C_VEL
LIN {X 0,Y 376.222,Z 166.615,A -85,B 0,C 180,E1 -12246.435,E2 -12246.435} C_VEL
LIN {X 0,Y 376.107,Z 166.629,A -85,B 0,C 180,E1 -12249.682,E2 -12249.682} C_VEL
LIN {X 0,Y 376.084,Z 166.639,A -85,B 0,C 180,E1 -12253.658,E2 -12253.658} C_VEL
LIN {X 0,Y 376.027,Z 166.635,A -85,B 0,C 180,E1 -12257.4,E2 -12257.4} C_VEL
LIN {X 0,Y 375.974,Z 166.651,A -85,B 0,C 180,E1 -12260.832,E2 -12260.832} C_VEL
LIN {X 0,Y 375.982,Z 166.639,A -85,B 0,C 180,E1 -12264.282,E2 -12264.282} C_VEL
LIN {X 0,Y 376.015,Z 166.646,A -85,B 0,C 180,E1 -12266.652,E2 -12266.652} C_VEL
LIN {X 0,Y 375.96,Z 166.647,A -85,B 0,C 180,E1 -12270.313,E2 -12270.313} C_VEL
LIN {X 0,Y 375.956,Z 166.645,A -85,B 0,C 180,E1 -12274.112,E2 -12274.112} C_VEL
LIN {X 0,Y 375.949,Z 166.624,A -85,B 0,C 180,E1 -12276.742,E2 -12276.742} C_VEL
LIN {X 0,Y 375.985,Z 166.648,A -85,B 0,C 180,E1 -12279.971,E2 -12279.971} C_VEL
LIN {X 0,Y 375.927,Z 166.653,A -85,B 0,C 180,E1 -12283.767,E2 -12283.767} C_VEL
LIN {X 0,Y 375.932,Z 166.653,A -85,B 0,C 180,E1 -12286.811,E2 -12286.811} C_VEL
LIN {X 0,Y 375.937,Z 166.645,A -85,B 0,C 180,E1 -12290.535,E2 -12290.535} C_VEL
LIN {X 0,Y 375.962,Z 166.654,A -85,B 0,C 180,E1 -12293.496,E2 -12293.496} C_VEL
LIN {X 0,Y 375.96,Z 166.643,A -85,B 0,C 180,E1 -12295.889,E2 -12295.889} C_VEL
LIN {X 0,Y 375.962,Z 166.646,A -85,B 0,C 180,E1 -12299.687,E2 -12299.687} C_VEL
LIN {X 0,Y 375.967,Z 166.735,A -85,B 0,C 180,E1 -12301.923,E2 -12301.923} C_VEL
LIN {X 0,Y 377.89,Z 175.719,A -85,B 0,C 180,E1 -12304.38,E2 -12304.38} C_VEL
LIN {X 0,Y 379.332,Z 184.077,A -85,B 0,C 180,E1 -12306.526,E2 -12306.526} C_VEL
LIN {X 0,Y 378.499,Z 193.543,A -85,B 0,C 180,E1 -12308.718,E2 -12308.718} C_VEL
LIN {X 0,Y 379.552,Z 199.321,A -85,B 0,C 180,E1 -12308.945,E2 -12308.945} C_VEL
LIN {X 0,Y 383.6,Z 222.385,A -85,B 0,C 180,E1 -12309.629,E2 -12309.629} C_VEL
LIN {X 0,Y 382.481,Z 301.466,A -85,B 0,C 180,E1 -12311.139,E2 -12311.139} C_VEL
LIN {X 0,Y 381.87,Z 314.671,A -85,B 0,C 180,E1 -12311.594,E2 -12311.594} C_VEL
LIN {X 0,Y 381.097,Z 326.791,A -85,B 0,C 180,E1 -12312.216,E2 -12312.216} C_VEL
LIN {X 0,Y 380.17,Z 339.021,A -85,B 0,C 180,E1 -12313.072,E2 -12313.072} C_VEL
LIN {X 0,Y 379.148,Z 350.59,A -85,B 0,C 180,E1 -12314.133,E2 -12314.133} C_VEL
LIN {X 0,Y 378.157,Z 361.334,A -85,B 0,C 180,E1 -12315.375,E2 -12315.375} C_VEL
LIN {X 0,Y 377.209,Z 371.182,A -85,B 0,C 180,E1 -12316.807,E2 -12316.807} C_VEL
LIN {X 0,Y 376.225,Z 380.09,A -85,B 0,C 180,E1 -12318.415,E2 -12318.415} C_VEL
LIN {X 0,Y 375.572,Z 387.257,A -85,B 0,C 180,E1 -12320.032,E2 -12320.032} C_VEL
LIN {X 0,Y 375.005,Z 393.782,A -85,B 0,C 180,E1 -12321.92,E2 -12321.92} C_VEL
LIN {X 0,Y 374.676,Z 398.702,A -85,B 0,C 180,E1 -12323.8,E2 -12323.8} C_VEL
LIN {X 0,Y 374.568,Z 402.234,A -85,B 0,C 180,E1 -12325.695,E2 -12325.695} C_VEL
LIN {X 0,Y 374.417,Z 404.611,A -85,B 0,C 180,E1 -12327.848,E2 -12327.848} C_VEL
LIN {X 0,Y 374.452,Z 405.216,A -85,B 0,C 180,E1 -12328.924,E2 -12328.924} C_VEL
LIN {X 0,Y 374.473,Z 405.429,A -85,B 0,C 180,E1 -12330,E2 -12330} C_VEL
LIN {X 0,Y 374.452,Z 405.212,A -85,B 0,C 180,E1 -12331.075,E2 -12331.075} C_VEL
LIN {X 0,Y 374.442,Z 403.614,A -85,B 0,C 180,E1 -12333.227,E2 -12333.227} C_VEL
LIN {X 0,Y 374.568,Z 402.223,A -85,B 0,C 180,E1 -12334.304,E2 -12334.304} C_VEL
LIN {X 0,Y 374.676,Z 398.679,A -85,B 0,C 180,E1 -12336.199,E2 -12336.199} C_VEL
LIN {X 0,Y 375.006,Z 393.75,A -85,B 0,C 180,E1 -12338.079,E2 -12338.079} C_VEL
LIN {X 0,Y 375.461,Z 388.239,A -85,B 0,C 180,E1 -12339.698,E2 -12339.698} C_VEL
LIN {X 0,Y 376.121,Z 381.358,A -85,B 0,C 180,E1 -12341.314,E2 -12341.314} C_VEL
LIN {X 0,Y 377.039,Z 372.747,A -85,B 0,C 180,E1 -12342.924,E2 -12342.924} C_VEL
LIN {X 0,Y 378.023,Z 362.631,A -85,B 0,C 180,E1 -12344.441,E2 -12344.441} C_VEL
LIN {X 0,Y 378.995,Z 352.163,A -85,B 0,C 180,E1 -12345.694,E2 -12345.694} C_VEL
LIN {X 0,Y 379.982,Z 340.475,A -85,B 0,C 180,E1 -12346.797,E2 -12346.797} C_VEL
LIN {X 0,Y 380.957,Z 328.75,A -85,B 0,C 180,E1 -12347.652,E2 -12347.652} C_VEL
LIN {X 0,Y 381.761,Z 315.931,A -85,B 0,C 180,E1 -12348.341,E2 -12348.341} C_VEL
LIN {X 0,Y 382.357,Z 302.221,A -85,B 0,C 180,E1 -12348.832,E2 -12348.832} C_VEL
LIN {X 0,Y 382.947,Z 270.589,A -85,B 0,C 180,E1 -12349.453,E2 -12349.453} C_VEL
LIN {X 0,Y 383.529,Z 221.773,A -85,B 0,C 180,E1 -12350.374,E2 -12350.374} C_VEL
LIN {X 0,Y 378.562,Z 194.047,A -85,B 0,C 180,E1 -12351.22,E2 -12351.22} C_VEL
LIN {X 0,Y 378.538,Z 193.009,A -85,B 0,C 180,E1 -12351.368,E2 -12351.368} C_VEL
LIN {X 0,Y 379.293,Z 184.021,A -85,B 0,C 180,E1 -12353.476,E2 -12353.476} C_VEL
LIN {X 0,Y 377.852,Z 175.659,A -85,B 0,C 180,E1 -12355.622,E2 -12355.622} C_VEL
LIN {X 0,Y 376.017,Z 166.931,A -85,B 0,C 180,E1 -12357.964,E2 -12357.964} C_VEL
LIN {X 0,Y 375.954,Z 166.644,A -85,B 0,C 180,E1 -12358.525,E2 -12358.525} C_VEL
LIN {X 0,Y 375.954,Z 166.654,A -85,B 0,C 180,E1 -12361.561,E2 -12361.561} C_VEL
LIN {X 0,Y 375.953,Z 166.656,A -85,B 0,C 180,E1 -12365.414,E2 -12365.414} C_VEL
LIN {X 0,Y 375.933,Z 166.637,A -85,B 0,C 180,E1 -12368.262,E2 -12368.262} C_VEL
LIN {X 0,Y 375.924,Z 166.657,A -85,B 0,C 180,E1 -12371.599,E2 -12371.599} C_VEL
LIN {X 0,Y 375.921,Z 166.658,A -85,B 0,C 180,E1 -12375.268,E2 -12375.268} C_VEL
LIN {X 0,Y 375.927,Z 166.655,A -85,B 0,C 180,E1 -12378.398,E2 -12378.398} C_VEL
LIN {X 0,Y 375.964,Z 166.636,A -85,B 0,C 180,E1 -12381.729,E2 -12381.729} C_VEL
LIN {X 0,Y 375.971,Z 166.638,A -85,B 0,C 180,E1 -12385.332,E2 -12385.332} C_VEL
LIN {X 0,Y 375.948,Z 166.655,A -85,B 0,C 180,E1 -12388.437,E2 -12388.437} C_VEL
LIN {X 0,Y 375.973,Z 166.648,A -85,B 0,C 180,E1 -12392.139,E2 -12392.139} C_VEL
LIN {X 0,Y 375.995,Z 166.649,A -85,B 0,C 180,E1 -12394.538,E2 -12394.538} C_VEL
LIN {X 0,Y 375.946,Z 166.652,A -85,B 0,C 180,E1 -12398.045,E2 -12398.045} C_VEL
LIN {X 0,Y 375.991,Z 166.637,A -85,B 0,C 180,E1 -12401.472,E2 -12401.472} C_VEL
LIN {X 0,Y 376.048,Z 166.645,A -85,B 0,C 180,E1 -12404.832,E2 -12404.832} C_VEL
LIN {X 0,Y 376.048,Z 166.632,A -85,B 0,C 180,E1 -12408.137,E2 -12408.137} C_VEL
LIN {X 0,Y 376.208,Z 166.621,A -85,B 0,C 180,E1 -12411.919,E2 -12411.919} C_VEL
LIN {X 0,Y 376.156,Z 166.617,A -85,B 0,C 180,E1 -12414.64,E2 -12414.64} C_VEL
LIN {X 0,Y 376.339,Z 166.603,A -85,B 0,C 180,E1 -12417.86,E2 -12417.86} C_VEL
LIN {X 0,Y 376.476,Z 166.588,A -85,B 0,C 180,E1 -12420,E2 -12420} C_VEL
LIN {X 0,Y 376.17,Z 166.618,A -85,B 0,C 180,E1 -12423.213,E2 -12423.213} C_VEL
LIN {X 0,Y 376.216,Z 166.619,A -85,B 0,C 180,E1 -12426.698,E2 -12426.698} C_VEL
LIN {X 0,Y 376.194,Z 166.611,A -85,B 0,C 180,E1 -12428.595,E2 -12428.595} C_VEL
LIN {X 0,Y 376.038,Z 166.64,A -85,B 0,C 180,E1 -12431.864,E2 -12431.864} C_VEL
LIN {X 0,Y 376.047,Z 166.63,A -85,B 0,C 180,E1 -12435.168,E2 -12435.168} C_VEL
LIN {X 0,Y 376.013,Z 166.648,A -85,B 0,C 180,E1 -12438.527,E2 -12438.527} C_VEL
LIN {X 0,Y 375.953,Z 166.645,A -85,B 0,C 180,E1 -12441.955,E2 -12441.955} C_VEL
LIN {X 0,Y 375.997,Z 166.647,A -85,B 0,C 180,E1 -12445.462,E2 -12445.462} C_VEL
LIN {X 0,Y 375.961,Z 166.649,A -85,B 0,C 180,E1 -12449.08,E2 -12449.08} C_VEL
LIN {X 0,Y 375.941,Z 166.644,A -85,B 0,C 180,E1 -12452.83,E2 -12452.83} C_VEL
LIN {X 0,Y 375.949,Z 166.619,A -85,B 0,C 180,E1 -12455.417,E2 -12455.417} C_VEL
LIN {X 0,Y 375.967,Z 166.65,A -85,B 0,C 180,E1 -12458.271,E2 -12458.271} C_VEL
LIN {X 0,Y 375.928,Z 166.649,A -85,B 0,C 180,E1 -12461.602,E2 -12461.602} C_VEL
LIN {X 0,Y 375.921,Z 166.649,A -85,B 0,C 180,E1 -12465.27,E2 -12465.27} C_VEL
LIN {X 0,Y 375.929,Z 166.649,A -85,B 0,C 180,E1 -12468.401,E2 -12468.401} C_VEL
LIN {X 0,Y 375.968,Z 166.645,A -85,B 0,C 180,E1 -12471.731,E2 -12471.731} C_VEL
LIN {X 0,Y 375.977,Z 166.639,A -85,B 0,C 180,E1 -12475.334,E2 -12475.334} C_VEL
LIN {X 0,Y 375.955,Z 166.646,A -85,B 0,C 180,E1 -12478.439,E2 -12478.439} C_VEL
LIN {X 0,Y 375.982,Z 166.648,A -85,B 0,C 180,E1 -12482.141,E2 -12482.141} C_VEL
LIN {X 0,Y 376.075,Z 166.886,A -85,B 0,C 180,E1 -12483.486,E2 -12483.486} C_VEL
LIN {X 0,Y 378.463,Z 178.949,A -85,B 0,C 180,E1 -12486.759,E2 -12486.759} C_VEL
LIN {X 0,Y 378.951,Z 182.39,A -85,B 0,C 180,E1 -12487.652,E2 -12487.652} C_VEL
LIN {X 0,Y 378.663,Z 187.349,A -85,B 0,C 180,E1 -12488.803,E2 -12488.803} C_VEL
LIN {X 0,Y 380.974,Z 198.881,A -85,B 0,C 180,E1 -12489.206,E2 -12489.206} C_VEL
LIN {X 0,Y 383.692,Z 213.916,A -85,B 0,C 180,E1 -12489.655,E2 -12489.655} C_VEL
LIN {X 0,Y 382.553,Z 294.087,A -85,B 0,C 180,E1 -12491.178,E2 -12491.178} C_VEL
LIN {X 0,Y 382.035,Z 306.79,A -85,B 0,C 180,E1 -12491.603,E2 -12491.603} C_VEL
LIN {X 0,Y 381.263,Z 320.351,A -85,B 0,C 180,E1 -12492.294,E2 -12492.294} C_VEL
LIN {X 0,Y 380.386,Z 331.715,A -85,B 0,C 180,E1 -12493.083,E2 -12493.083} C_VEL
LIN {X 0,Y 379.41,Z 343.247,A -85,B 0,C 180,E1 -12494.13,E2 -12494.13} C_VEL
LIN {X 0,Y 378.549,Z 353.868,A -85,B 0,C 180,E1 -12495.348,E2 -12495.348} C_VEL
LIN {X 0,Y 377.656,Z 362.433,A -85,B 0,C 180,E1 -12496.549,E2 -12496.549} C_VEL
LIN {X 0,Y 376.784,Z 370.325,A -85,B 0,C 180,E1 -12497.888,E2 -12497.888} C_VEL
LIN {X 0,Y 376.013,Z 378.04,A -85,B 0,C 180,E1 -12499.501,E2 -12499.501} C_VEL
LIN {X 0,Y 375.491,Z 383.306,A -85,B 0,C 180,E1 -12500.846,E2 -12500.846} C_VEL
LIN {X 0,Y 375.054,Z 388.418,A -85,B 0,C 180,E1 -12502.463,E2 -12502.463} C_VEL
LIN {X 0,Y 374.796,Z 392.128,A -85,B 0,C 180,E1 -12503.963,E2 -12503.963} C_VEL
LIN {X 0,Y 374.617,Z 395.321,A -85,B 0,C 180,E1 -12505.697,E2 -12505.697} C_VEL
LIN {X 0,Y 374.49,Z 396.728,A -85,B 0,C 180,E1 -12506.773,E2 -12506.773} C_VEL
LIN {X 0,Y 374.46,Z 398.343,A -85,B 0,C 180,E1 -12508.925,E2 -12508.925} C_VEL
LIN {X 0,Y 374.474,Z 398.577,A -85,B 0,C 180,E1 -12510,E2 -12510} C_VEL
LIN {X 0,Y 374.46,Z 398.387,A -85,B 0,C 180,E1 -12511.076,E2 -12511.076} C_VEL
LIN {X 0,Y 374.489,Z 396.829,A -85,B 0,C 180,E1 -12513.228,E2 -12513.228} C_VEL
LIN {X 0,Y 374.613,Z 395.466,A -85,B 0,C 180,E1 -12514.304,E2 -12514.304} C_VEL
LIN {X 0,Y 374.772,Z 392.427,A -85,B 0,C 180,E1 -12516.001,E2 -12516.001} C_VEL
LIN {X 0,Y 375.059,Z 388.685,A -85,B 0,C 180,E1 -12517.537,E2 -12517.537} C_VEL
LIN {X 0,Y 375.468,Z 383.652,A -85,B 0,C 180,E1 -12519.155,E2 -12519.155} C_VEL
LIN {X 0,Y 376.088,Z 377.317,A -85,B 0,C 180,E1 -12520.77,E2 -12520.77} C_VEL
LIN {X 0,Y 376.899,Z 369.389,A -85,B 0,C 180,E1 -12522.383,E2 -12522.383} C_VEL
LIN {X 0,Y 377.965,Z 359.529,A -85,B 0,C 180,E1 -12523.989,E2 -12523.989} C_VEL
LIN {X 0,Y 378.542,Z 353.995,A -85,B 0,C 180,E1 -12524.738,E2 -12524.738} C_VEL
LIN {X 0,Y 378.258,Z 349.534,A -85,B 0,C 180,E1 -12525.313,E2 -12525.313} C_VEL
LIN {X 0,Y 375.235,Z 338.961,A -85,B 0,C 180,E1 -12526.602,E2 -12526.602} C_VEL
LIN {X 0,Y 373.939,Z 332.475,A -85,B 0,C 180,E1 -12527.26,E2 -12527.26} C_VEL
LIN {X 0,Y 373.899,Z 328.987,A -85,B 0,C 180,E1 -12527.548,E2 -12527.548} C_VEL
LIN {X 0,Y 374.792,Z 316.424,A -85,B 0,C 180,E1 -12528.377,E2 -12528.377} C_VEL
LIN {X 0,Y 375.499,Z 303.444,A -85,B 0,C 180,E1 -12528.978,E2 -12528.978} C_VEL
LIN {X 0,Y 375.962,Z 291.052,A -85,B 0,C 180,E1 -12529.343,E2 -12529.343} C_VEL
LIN {X 0,Y 376.988,Z 214.293,A -85,B 0,C 180,E1 -12530.822,E2 -12530.822} C_VEL
LIN {X 0,Y 371.934,Z 188.124,A -85,B 0,C 180,E1 -12531.663,E2 -12531.663} C_VEL
LIN {X 0,Y 371.905,Z 186.793,A -85,B 0,C 180,E1 -12531.819,E2 -12531.819} C_VEL
LIN {X 0,Y 371.958,Z 182.886,A -85,B 0,C 180,E1 -12532.788,E2 -12532.788} C_VEL
LIN {X 0,Y 369.765,Z 171.362,A -85,B 0,C 180,E1 -12535.922,E2 -12535.922} C_VEL
LIN {X 0,Y 369.013,Z 167.579,A -85,B 0,C 180,E1 -12537.05,E2 -12537.05} C_VEL
LIN {X 0,Y 368.911,Z 167.522,A -85,B 0,C 180,E1 -12540.987,E2 -12540.987} C_VEL
LIN {X 0,Y 368.937,Z 167.515,A -85,B 0,C 180,E1 -12544.853,E2 -12544.853} C_VEL
LIN {X 0,Y 368.906,Z 167.523,A -85,B 0,C 180,E1 -12548.639,E2 -12548.639} C_VEL
LIN {X 0,Y 368.88,Z 167.529,A -85,B 0,C 180,E1 -12552.009,E2 -12552.009} C_VEL
LIN {X 0,Y 368.878,Z 167.527,A -85,B 0,C 180,E1 -12555.175,E2 -12555.175} C_VEL
LIN {X 0,Y 368.881,Z 167.52,A -85,B 0,C 180,E1 -12558.177,E2 -12558.177} C_VEL
LIN {X 0,Y 368.907,Z 167.531,A -85,B 0,C 180,E1 -12561.359,E2 -12561.359} C_VEL
LIN {X 0,Y 368.934,Z 167.49,A -85,B 0,C 180,E1 -12565.146,E2 -12565.146} C_VEL
LIN {X 0,Y 368.926,Z 167.527,A -85,B 0,C 180,E1 -12569.046,E2 -12569.046} C_VEL
LIN {X 0,Y 368.972,Z 167.52,A -85,B 0,C 180,E1 -12571.563,E2 -12571.563} C_VEL
LIN {X 0,Y 368.996,Z 167.52,A -85,B 0,C 180,E1 -12574.019,E2 -12574.019} C_VEL
LIN {X 0,Y 368.918,Z 167.522,A -85,B 0,C 180,E1 -12577.604,E2 -12577.604} C_VEL
LIN {X 0,Y 368.962,Z 167.524,A -85,B 0,C 180,E1 -12581.106,E2 -12581.106} C_VEL
LIN {X 0,Y 368.992,Z 167.508,A -85,B 0,C 180,E1 -12584.535,E2 -12584.535} C_VEL
LIN {X 0,Y 368.999,Z 167.52,A -85,B 0,C 180,E1 -12587.906,E2 -12587.906} C_VEL
LIN {X 0,Y 369.223,Z 167.482,A -85,B 0,C 180,E1 -12591.802,E2 -12591.802} C_VEL
LIN {X 0,Y 369.135,Z 167.5,A -85,B 0,C 180,E1 -12594.537,E2 -12594.537} C_VEL
LIN {X 0,Y 369.309,Z 167.469,A -85,B 0,C 180,E1 -12597.819,E2 -12597.819} C_VEL
LIN {X 0,Y 369.45,Z 167.464,A -85,B 0,C 180,E1 -12600,E2 -12600} C_VEL
LIN {X 0,Y 369.31,Z 167.478,A -85,B 0,C 180,E1 -12602.181,E2 -12602.181} C_VEL
LIN {X 0,Y 369.181,Z 167.492,A -85,B 0,C 180,E1 -12606.559,E2 -12606.559} C_VEL
LIN {X 0,Y 369.057,Z 167.506,A -85,B 0,C 180,E1 -12609.869,E2 -12609.869} C_VEL
LIN {X 0,Y 369.032,Z 167.516,A -85,B 0,C 180,E1 -12613.772,E2 -12613.772} C_VEL
LIN {X 0,Y 368.986,Z 167.51,A -85,B 0,C 180,E1 -12617.743,E2 -12617.743} C_VEL
LIN {X 0,Y 368.905,Z 167.535,A -85,B 0,C 180,E1 -12621.221,E2 -12621.221} C_VEL
LIN {X 0,Y 368.949,Z 167.518,A -85,B 0,C 180,E1 -12624.776,E2 -12624.776} C_VEL
LIN {X 0,Y 368.959,Z 167.527,A -85,B 0,C 180,E1 -12627.204,E2 -12627.204} C_VEL
LIN {X 0,Y 368.926,Z 167.528,A -85,B 0,C 180,E1 -12630.954,E2 -12630.954} C_VEL
LIN {X 0,Y 368.925,Z 167.508,A -85,B 0,C 180,E1 -12635.002,E2 -12635.002} C_VEL
LIN {X 0,Y 368.903,Z 167.519,A -85,B 0,C 180,E1 -12638.64,E2 -12638.64} C_VEL
LIN {X 0,Y 368.877,Z 167.531,A -85,B 0,C 180,E1 -12642.01,E2 -12642.01} C_VEL
LIN {X 0,Y 368.877,Z 167.537,A -85,B 0,C 180,E1 -12645.176,E2 -12645.176} C_VEL
LIN {X 0,Y 368.87,Z 167.535,A -85,B 0,C 180,E1 -12648.176,E2 -12648.176} C_VEL
LIN {X 0,Y 368.876,Z 167.516,A -85,B 0,C 180,E1 -12651.366,E2 -12651.366} C_VEL
LIN {X 0,Y 368.936,Z 167.522,A -85,B 0,C 180,E1 -12655.147,E2 -12655.147} C_VEL
LIN {X 0,Y 368.93,Z 167.522,A -85,B 0,C 180,E1 -12659.047,E2 -12659.047} C_VEL
LIN {X 0,Y 368.954,Z 167.702,A -85,B 0,C 180,E1 -12661.64,E2 -12661.64} C_VEL
LIN {X 0,Y 371.349,Z 179.134,A -85,B 0,C 180,E1 -12664.772,E2 -12664.772} C_VEL
LIN {X 0,Y 372.376,Z 185.202,A -85,B 0,C 180,E1 -12666.356,E2 -12666.356} C_VEL
LIN {X 0,Y 371.656,Z 193.64,A -85,B 0,C 180,E1 -12668.325,E2 -12668.325} C_VEL
LIN {X 0,Y 374.845,Z 210.527,A -85,B 0,C 180,E1 -12668.894,E2 -12668.894} C_VEL
LIN {X 0,Y 377.028,Z 224.273,A -85,B 0,C 180,E1 -12669.296,E2 -12669.296} C_VEL
LIN {X 0,Y 375.787,Z 301.414,A -85,B 0,C 180,E1 -12670.79,E2 -12670.79} C_VEL
LIN {X 0,Y 375.154,Z 314.614,A -85,B 0,C 180,E1 -12671.252,E2 -12671.252} C_VEL
LIN {X 0,Y 374.344,Z 326.732,A -85,B 0,C 180,E1 -12671.884,E2 -12671.884} C_VEL
LIN {X 0,Y 373.386,Z 338.96,A -85,B 0,C 180,E1 -12672.755,E2 -12672.755} C_VEL
LIN {X 0,Y 372.311,Z 350.526,A -85,B 0,C 180,E1 -12673.833,E2 -12673.833} C_VEL
LIN {X 0,Y 371.346,Z 360.603,A -85,B 0,C 180,E1 -12675.013,E2 -12675.013} C_VEL
LIN {X 0,Y 370.495,Z 369.449,A -85,B 0,C 180,E1 -12676.284,E2 -12676.284} C_VEL
LIN {X 0,Y 369.562,Z 377.298,A -85,B 0,C 180,E1 -12677.646,E2 -12677.646} C_VEL
LIN {X 0,Y 368.789,Z 384.963,A -85,B 0,C 180,E1 -12679.292,E2 -12679.292} C_VEL
LIN {X 0,Y 368.084,Z 392.03,A -85,B 0,C 180,E1 -12681.214,E2 -12681.214} C_VEL
LIN {X 0,Y 367.702,Z 396.729,A -85,B 0,C 180,E1 -12682.863,E2 -12682.863} C_VEL
LIN {X 0,Y 367.528,Z 400.319,A -85,B 0,C 180,E1 -12684.513,E2 -12684.513} C_VEL
LIN {X 0,Y 367.477,Z 402.17,A -85,B 0,C 180,E1 -12685.612,E2 -12685.612} C_VEL
LIN {X 0,Y 367.32,Z 404.546,A -85,B 0,C 180,E1 -12687.807,E2 -12687.807} C_VEL
LIN {X 0,Y 367.35,Z 405.151,A -85,B 0,C 180,E1 -12688.903,E2 -12688.903} C_VEL
LIN {X 0,Y 367.374,Z 405.364,A -85,B 0,C 180,E1 -12690,E2 -12690} C_VEL
LIN {X 0,Y 367.35,Z 405.147,A -85,B 0,C 180,E1 -12691.096,E2 -12691.096} C_VEL
LIN {X 0,Y 367.363,Z 403.548,A -85,B 0,C 180,E1 -12693.29,E2 -12693.29} C_VEL
LIN {X 0,Y 367.476,Z 402.157,A -85,B 0,C 180,E1 -12694.387,E2 -12694.387} C_VEL
LIN {X 0,Y 367.584,Z 398.956,A -85,B 0,C 180,E1 -12696.167,E2 -12696.167} C_VEL
LIN {X 0,Y 367.849,Z 395.272,A -85,B 0,C 180,E1 -12697.685,E2 -12697.685} C_VEL
LIN {X 0,Y 368.335,Z 389.181,A -85,B 0,C 180,E1 -12699.61,E2 -12699.61} C_VEL
LIN {X 0,Y 369.017,Z 382.525,A -85,B 0,C 180,E1 -12701.256,E2 -12701.256} C_VEL
LIN {X 0,Y 369.926,Z 374.264,A -85,B 0,C 180,E1 -12702.898,E2 -12702.898} C_VEL
LIN {X 0,Y 370.837,Z 365.793,A -85,B 0,C 180,E1 -12704.262,E2 -12704.262} C_VEL
LIN {X 0,Y 371.813,Z 355.321,A -85,B 0,C 180,E1 -12705.625,E2 -12705.625} C_VEL
LIN {X 0,Y 372.93,Z 343.532,A -85,B 0,C 180,E1 -12706.842,E2 -12706.842} C_VEL
LIN {X 0,Y 373.974,Z 331.664,A -85,B 0,C 180,E1 -12707.78,E2 -12707.78} C_VEL
LIN {X 0,Y 374.889,Z 319.311,A -85,B 0,C 180,E1 -12708.512,E2 -12708.512} C_VEL
LIN {X 0,Y 375.519,Z 306.61,A -85,B 0,C 180,E1 -12709.046,E2 -12709.046} C_VEL
LIN {X 0,Y 375.974,Z 293.261,A -85,B 0,C 180,E1 -12709.377,E2 -12709.377} C_VEL
LIN {X 0,Y 376.93,Z 222.965,A -85,B 0,C 180,E1 -12710.722,E2 -12710.722} C_VEL
LIN {X 0,Y 371.949,Z 195.383,A -85,B 0,C 180,E1 -12711.571,E2 -12711.571} C_VEL
LIN {X 0,Y 371.659,Z 193.539,A -85,B 0,C 180,E1 -12711.673,E2 -12711.673} C_VEL
LIN {X 0,Y 372.357,Z 185.143,A -85,B 0,C 180,E1 -12713.645,E2 -12713.645} C_VEL
LIN {X 0,Y 370.857,Z 176.782,A -85,B 0,C 180,E1 -12715.839,E2 -12715.839} C_VEL
LIN {X 0,Y 368.93,Z 167.604,A -85,B 0,C 180,E1 -12718.4,E2 -12718.4} C_VEL
LIN {X 0,Y 368.907,Z 167.526,A -85,B 0,C 180,E1 -12720.986,E2 -12720.986} C_VEL
LIN {X 0,Y 368.932,Z 167.523,A -85,B 0,C 180,E1 -12724.852,E2 -12724.852} C_VEL
LIN {X 0,Y 368.874,Z 167.517,A -85,B 0,C 180,E1 -12728.633,E2 -12728.633} C_VEL
LIN {X 0,Y 368.872,Z 167.534,A -85,B 0,C 180,E1 -12732.008,E2 -12732.008} C_VEL
LIN {X 0,Y 368.874,Z 167.537,A -85,B 0,C 180,E1 -12735.175,E2 -12735.175} C_VEL
LIN {X 0,Y 368.876,Z 167.532,A -85,B 0,C 180,E1 -12738.176,E2 -12738.176} C_VEL
LIN {X 0,Y 368.899,Z 167.518,A -85,B 0,C 180,E1 -12741.359,E2 -12741.359} C_VEL
LIN {X 0,Y 368.928,Z 167.512,A -85,B 0,C 180,E1 -12745.145,E2 -12745.145} C_VEL
LIN {X 0,Y 368.921,Z 167.528,A -85,B 0,C 180,E1 -12749.046,E2 -12749.046} C_VEL
